C01820=1176.293,412.482,-85.837,-176.041,9.220,148.722
C01821=1176.297,412.234,-85.801,-176.041,9.217,148.722
C01822=1176.301,411.988,-85.765,-176.040,9.216,148.721
C01823=1176.305,411.740,-85.728,-176.040,9.215,148.721
C01824=1176.309,411.492,-85.693,-176.040,9.212,148.720
C01825=1176.313,411.245,-85.656,-176.040,9.210,148.719
C01826=1176.317,410.998,-85.621,-176.040,9.208,148.719
C01827=1176.321,410.750,-85.584,-176.039,9.206,148.718
C01828=1176.324,410.503,-85.548,-176.039,9.204,148.718
C01829=1176.328,410.255,-85.513,-176.039,9.202,148.717
C01830=1176.333,410.008,-85.476,-176.039,9.200,148.717
C01831=1176.336,409.761,-85.440,-176.038,9.198,148.716
C01832=1176.340,409.513,-85.404,-176.038,9.196,148.715
C01833=1176.344,409.266,-85.368,-176.038,9.195,148.715
C01834=1176.348,409.018,-85.332,-176.038,9.192,148.714
C01835=1176.352,408.771,-85.296,-176.038,9.191,148.714
C01836=1176.356,408.525,-85.260,-176.038,9.188,148.713
C01837=1176.360,408.277,-85.224,-176.038,9.186,148.713
C01838=1176.364,408.029,-85.188,-176.037,9.184,148.712
C01839=1176.368,407.782,-85.152,-176.037,9.182,148.711
C01840=1176.371,407.535,-85.116,-176.037,9.180,148.711
C01841=1176.375,407.287,-85.081,-176.037,9.178,148.710
C01842=1176.379,407.040,-85.044,-176.036,9.176,148.710
C01843=1176.383,406.792,-85.008,-176.036,9.174,148.709
C01844=1176.387,406.545,-84.972,-176.036,9.171,148.708
C01845=1176.391,406.297,-84.936,-176.036,9.170,148.708
C01846=1176.395,406.050,-84.900,-176.036,9.167,148.707
C01847=1176.399,405.803,-84.864,-176.036,9.166,148.707
C01848=1176.403,405.556,-84.829,-176.035,9.163,148.706
C01849=1176.407,405.308,-84.792,-176.035,9.161,148.705
C01850=1176.411,405.061,-84.756,-176.035,9.159,148.705
C01851=1176.414,404.813,-84.721,-176.035,9.157,148.704
C01852=1176.418,404.566,-84.684,-176.035,9.155,148.704
C01853=1176.422,404.319,-84.648,-176.034,9.153,148.703
C01854=1176.427,404.071,-84.612,-176.034,9.150,148.702
C01855=1176.430,403.823,-84.577,-176.034,9.148,148.702
C01856=1176.434,403.576,-84.541,-176.034,9.145,148.701
C01857=1176.439,403.329,-84.505,-176.034,9.144,148.701
C01858=1176.442,403.082,-84.469,-176.034,9.141,148.700
C01859=1176.446,402.835,-84.432,-176.034,9.139,148.699
C01860=1176.450,402.587,-84.397,-176.034,9.137,148.699
C01861=1176.454,402.340,-84.361,-176.033,9.135,148.698
C01862=1176.458,402.092,-84.325,-176.033,9.132,148.697
C01863=1176.461,401.845,-84.289,-176.033,9.130,148.697
C01864=1176.465,401.597,-84.253,-176.033,9.127,148.696
C01865=1176.470,401.350,-84.218,-176.032,9.126,148.695
C01866=1176.474,401.103,-84.182,-176.033,9.123,148.695
C01867=1176.477,400.855,-84.146,-176.033,9.121,148.694
C01868=1176.481,400.608,-84.110,-176.032,9.118,148.693
C01869=1176.485,400.361,-84.074,-176.033,9.116,148.693
C01870=1176.490,400.113,-84.038,-176.033,9.113,148.692
C01871=1176.493,399.865,-84.002,-176.032,9.111,148.691
C01872=1176.497,399.618,-83.966,-176.032,9.109,148.691
C01873=1176.502,399.371,-83.930,-176.032,9.107,148.690
C01874=1176.505,399.124,-83.895,-176.032,9.104,148.689
C01875=1176.509,398.876,-83.859,-176.032,9.102,148.689
C01876=1176.513,398.629,-83.823,-176.032,9.099,148.688
C01877=1176.517,398.382,-83.787,-176.032,9.097,148.688
C01878=1176.520,398.134,-83.751,-176.032,9.094,148.687
C01879=1176.525,397.886,-83.715,-176.032,9.092,148.686
C01880=1176.529,397.640,-83.680,-176.032,9.089,148.686
C01881=1176.533,397.392,-83.644,-176.031,9.087,148.685
C01882=1176.537,397.144,-83.608,-176.031,9.084,148.684
C01883=1176.540,396.897,-83.572,-176.032,9.082,148.684
C01884=1176.544,396.650,-83.536,-176.031,9.080,148.683
C01885=1176.548,396.402,-83.501,-176.031,9.077,148.682
C01886=1176.552,396.155,-83.465,-176.032,9.075,148.682
C01887=1176.556,395.908,-83.430,-176.032,9.071,148.681
C01888=1176.560,395.660,-83.394,-176.032,9.069,148.680
C01889=1176.564,395.412,-83.358,-176.032,9.066,148.679
C01890=1176.568,395.166,-83.322,-176.032,9.064,148.679
C01891=1176.571,394.918,-83.286,-176.032,9.061,148.678
C01892=1176.576,394.670,-83.250,-176.032,9.059,148.678
C01893=1176.580,394.423,-83.215,-176.031,9.056,148.677
C01894=1176.584,394.176,-83.179,-176.032,9.053,148.676
C01895=1176.587,393.928,-83.144,-176.032,9.051,148.675
C01896=1176.592,393.681,-83.107,-176.032,9.048,148.675
C01897=1176.596,393.433,-83.072,-176.032,9.045,148.674
C01898=1176.599,393.186,-83.036,-176.033,9.042,148.673
C01899=1176.603,392.939,-83.000,-176.032,9.040,148.673
C01900=1176.608,392.692,-82.964,-176.032,9.037,148.672
C01901=1176.611,392.444,-82.929,-176.033,9.034,148.671
C01902=1176.616,392.159,-82.888,-176.032,9.031,148.671
C01903=1176.620,391.875,-82.847,-176.033,9.028,148.670
C01904=1176.625,391.591,-82.806,-176.033,9.024,148.669
C01905=1176.629,391.307,-82.765,-176.034,9.021,148.668
C01906=1176.633,391.059,-82.729,-176.033,9.018,148.667
C01907=1176.637,390.811,-82.693,-176.034,9.016,148.667
C01908=1176.641,390.564,-82.658,-176.034,9.013,148.666
C01909=1176.645,390.317,-82.622,-176.034,9.010,148.665
C01910=1176.649,390.070,-82.587,-176.035,9.007,148.665
C01911=1176.653,389.822,-82.551,-176.035,9.005,148.664
C01912=1176.657,389.574,-82.515,-176.035,9.001,148.663
C01913=1176.661,389.327,-82.480,-176.036,8.998,148.663
C01914=1176.665,389.080,-82.444,-176.036,8.996,148.662
C01915=1176.668,388.832,-82.409,-176.037,8.992,148.662
C01916=1176.672,388.585,-82.373,-176.036,8.990,148.661
C01917=1176.677,388.337,-82.337,-176.037,8.986,148.660
C01918=1176.680,388.090,-82.302,-176.038,8.983,148.659
C01919=1176.684,387.843,-82.266,-176.037,8.981,148.659
C01920=1176.688,387.595,-82.231,-176.038,8.978,148.658
C01921=1176.692,387.348,-82.195,-176.039,8.974,148.657
C01922=1176.696,387.100,-82.159,-176.039,8.971,148.657
C01923=1176.700,386.853,-82.124,-176.039,8.969,148.656
C01924=1176.704,386.605,-82.089,-176.040,8.966,148.656
C01925=1176.708,386.358,-82.054,-176.041,8.962,148.655
C01926=1176.712,386.110,-82.018,-176.041,8.959,148.654
C01927=1176.715,385.863,-81.983,-176.042,8.956,148.653
C01928=1176.720,385.616,-81.947,-176.043,8.953,148.653
C01929=1176.724,385.368,-81.911,-176.043,8.949,148.652
C01930=1176.728,385.120,-81.876,-176.043,8.947,148.651
C01931=1176.731,384.873,-81.840,-176.044,8.944,148.651
C01932=1176.736,384.626,-81.805,-176.045,8.940,148.650
C01933=1176.740,384.378,-81.770,-176.045,8.937,148.650
C01934=1176.743,384.131,-81.735,-176.046,8.934,148.649
C01935=1176.747,383.883,-81.699,-176.047,8.931,148.648
C01936=1176.751,383.636,-81.664,-176.047,8.928,148.648
C01937=1176.756,383.388,-81.628,-176.048,8.924,148.647
C01938=1176.759,383.141,-81.592,-176.049,8.920,148.646
C01939=1176.764,382.894,-81.558,-176.050,8.917,148.646
C01940=1176.768,382.646,-81.522,-176.050,8.914,148.645
C01941=1176.771,382.399,-81.487,-176.051,8.911,148.644
C01942=1176.775,382.151,-81.451,-176.052,8.908,148.644
C01943=1176.779,381.904,-81.416,-176.053,8.905,148.643
C01944=1176.783,381.656,-81.381,-176.054,8.901,148.642
C01945=1176.787,381.409,-81.345,-176.055,8.897,148.642
C01946=1176.791,381.162,-81.310,-176.056,8.894,148.641
C01947=1176.795,380.914,-81.275,-176.056,8.891,148.641
C01948=1176.799,380.666,-81.240,-176.057,8.888,148.640
C01949=1176.803,380.419,-81.205,-176.059,8.884,148.639
C01950=1176.807,380.172,-81.169,-176.059,8.881,148.639
C01951=1176.811,379.924,-81.134,-176.060,8.878,148.638
C01952=1176.815,379.676,-81.098,-176.062,8.874,148.638
C01953=1176.819,379.429,-81.063,-176.062,8.871,148.637
C01954=1176.823,379.181,-81.028,-176.063,8.868,148.636
C01955=1176.827,378.934,-80.993,-176.065,8.864,148.636
C01956=1176.831,378.687,-80.957,-176.066,8.861,148.635
C01957=1176.835,378.439,-80.923,-176.067,8.857,148.635
C01958=1176.839,378.191,-80.887,-176.068,8.854,148.634
C01959=1176.843,377.944,-80.852,-176.069,8.850,148.633
C01960=1176.847,377.696,-80.817,-176.070,8.847,148.633
C01961=1176.851,377.449,-80.782,-176.071,8.844,148.632
C01962=1176.854,377.202,-80.748,-176.072,8.840,148.632
C01963=1176.858,376.954,-80.712,-176.074,8.836,148.631
C01964=1176.862,376.707,-80.677,-176.074,8.833,148.630
C01965=1176.866,376.459,-80.642,-176.076,8.829,148.630
C01966=1176.870,376.212,-80.607,-176.077,8.826,148.629
C01967=1176.875,375.964,-80.572,-176.078,8.822,148.629
C01968=1176.878,375.717,-80.537,-176.079,8.819,148.628
C01969=1176.882,375.469,-80.502,-176.081,8.816,148.628
C01970=1176.886,375.222,-80.467,-176.083,8.812,148.627
C01971=1176.890,374.974,-80.432,-176.083,8.809,148.626
C01972=1176.895,374.727,-80.397,-176.085,8.805,148.626
C01973=1176.899,374.479,-80.362,-176.086,8.802,148.625
C01974=1176.902,374.231,-80.326,-176.087,8.798,148.625
C01975=1176.906,373.984,-80.292,-176.089,8.794,148.624
C01976=1176.910,373.737,-80.257,-176.090,8.791,148.624
C01977=1176.914,373.489,-80.222,-176.092,8.788,148.623
C01978=1176.918,373.242,-80.187,-176.093,8.784,148.623
C01979=1176.922,372.994,-80.152,-176.095,8.780,148.622
C01980=1176.927,372.746,-80.117,-176.096,8.777,148.622
C01981=1176.930,372.499,-80.082,-176.097,8.773,148.621
C01982=1176.934,372.252,-80.048,-176.099,8.769,148.621
C01983=1176.938,372.004,-80.012,-176.101,8.766,148.620
C01984=1176.942,371.756,-79.978,-176.102,8.763,148.620
C01985=1176.946,371.509,-79.943,-176.104,8.759,148.619
C01986=1176.950,371.261,-79.908,-176.105,8.755,148.619
C01987=1176.954,371.014,-79.874,-176.107,8.752,148.618
C01988=1176.958,370.766,-79.839,-176.109,8.748,148.618
C01989=1176.962,370.519,-79.804,-176.110,8.744,148.617
C01990=1176.966,370.271,-79.769,-176.111,8.741,148.617
C01991=1176.971,370.023,-79.734,-176.113,8.738,148.616
C01992=1176.974,369.776,-79.699,-176.115,8.734,148.616
C01993=1176.978,369.529,-79.665,-176.116,8.730,148.615
C01994=1176.982,369.281,-79.630,-176.118,8.727,148.615
C01995=1176.987,369.033,-79.596,-176.120,8.723,148.614
C01996=1176.990,368.786,-79.561,-176.122,8.719,148.614
C01997=1176.994,368.539,-79.526,-176.123,8.715,148.613
C01998=1176.998,368.291,-79.491,-176.125,8.712,148.613
C01999=1177.002,368.043,-79.458,-176.127,8.708,148.612
C02000=1177.006,367.795,-79.423,-176.129,8.705,148.612
C02001=1177.010,367.548,-79.388,-176.130,8.702,148.612
C02002=1177.014,367.300,-79.353,-176.132,8.698,148.611
C02003=1177.018,367.053,-79.319,-176.134,8.695,148.611
C02004=1177.022,366.805,-79.284,-176.136,8.691,148.610
C02005=1177.026,366.558,-79.250,-176.137,8.687,148.610
C02006=1177.030,366.276,-79.210,-176.140,8.683,148.609
C02007=1177.035,365.994,-79.171,-176.142,8.679,148.609
C02008=1177.040,365.712,-79.131,-176.144,8.675,148.609
C02009=1177.044,365.431,-79.093,-176.146,8.670,148.608
C02010=1177.048,365.182,-79.058,-176.148,8.667,148.608
C02011=1177.052,364.936,-79.024,-176.150,8.663,148.607
C02012=1177.056,364.688,-78.989,-176.152,8.660,148.607
C02013=1177.060,364.440,-78.955,-176.154,8.656,148.606
C02014=1177.064,364.193,-78.921,-176.156,8.652,148.606
C02015=1177.068,363.945,-78.886,-176.158,8.649,148.606
C02016=1177.072,363.698,-78.852,-176.160,8.645,148.605
C02017=1177.076,363.449,-78.818,-176.162,8.642,148.605
C02018=1177.080,363.202,-78.784,-176.163,8.638,148.604
C02019=1177.084,362.954,-78.749,-176.166,8.635,148.604
C02020=1177.089,362.707,-78.715,-176.167,8.631,148.604
C02021=1177.092,362.460,-78.681,-176.169,8.628,148.603
C02022=1177.096,362.211,-78.646,-176.171,8.624,148.603
C02023=1177.100,361.964,-78.612,-176.174,8.620,148.603
C02024=1177.104,361.716,-78.577,-176.176,8.616,148.602
C02025=1177.108,361.469,-78.543,-176.178,8.613,148.602
C02026=1177.113,361.222,-78.509,-176.180,8.609,148.602
C02027=1177.116,360.973,-78.475,-176.182,8.606,148.601
C02028=1177.121,360.726,-78.441,-176.184,8.602,148.601
C02029=1177.124,360.479,-78.407,-176.186,8.599,148.600
C02030=1177.128,360.231,-78.373,-176.188,8.595,148.600
C02031=1177.132,359.983,-78.338,-176.190,8.591,148.600
C02032=1177.136,359.735,-78.305,-176.193,8.588,148.600
C02033=1177.140,359.488,-78.270,-176.195,8.584,148.599
C02034=1177.144,359.241,-78.237,-176.197,8.581,148.599
C02035=1177.148,358.992,-78.202,-176.199,8.577,148.598
C02036=1177.152,358.745,-78.169,-176.201,8.574,148.598
C02037=1177.156,358.498,-78.135,-176.203,8.570,148.598
C02038=1177.160,358.249,-78.100,-176.206,8.566,148.598
C02039=1177.164,358.002,-78.067,-176.208,8.563,148.597
C02040=1177.169,357.754,-78.032,-176.210,8.559,148.597
C02041=1177.173,357.507,-77.998,-176.212,8.556,148.597
C02042=1177.176,357.259,-77.965,-176.214,8.552,148.596
C02043=1177.181,357.011,-77.930,-176.216,8.549,148.596
C02044=1177.185,356.764,-77.896,-176.218,8.546,148.596
C02045=1177.188,356.516,-77.863,-176.221,8.541,148.595
C02046=1177.193,356.268,-77.828,-176.223,8.538,148.595
C02047=1177.197,356.021,-77.795,-176.225,8.535,148.595
C02048=1177.201,355.774,-77.761,-176.227,8.531,148.594
C02049=1177.205,355.525,-77.727,-176.229,8.528,148.594
C02050=1177.209,355.278,-77.693,-176.232,8.524,148.594
C02051=1177.213,355.030,-77.660,-176.235,8.520,148.594
C02052=1177.217,354.783,-77.626,-176.236,8.517,148.593
C02053=1177.221,354.534,-77.592,-176.239,8.513,148.593
C02054=1177.225,354.287,-77.558,-176.241,8.510,148.593
C02055=1177.229,354.039,-77.525,-176.243,8.506,148.592
C02056=1177.234,353.792,-77.491,-176.245,8.503,148.592
C02057=1177.237,353.543,-77.457,-176.247,8.500,148.592
C02058=1177.241,353.296,-77.423,-176.250,8.496,148.592
C02059=1177.245,353.049,-77.390,-176.252,8.492,148.591
C02060=1177.250,352.801,-77.356,-176.254,8.489,148.591
C02061=1177.254,352.553,-77.323,-176.256,8.485,148.591
C02062=1177.257,352.305,-77.289,-176.259,8.482,148.591
C02063=1177.261,352.058,-77.255,-176.261,8.479,148.590
C02064=1177.265,351.810,-77.222,-176.263,8.475,148.590
C02065=1177.270,351.562,-77.188,-176.265,8.472,148.590
C02066=1177.274,351.315,-77.155,-176.268,8.468,148.589
C02067=1177.278,351.067,-77.121,-176.270,8.464,148.589
C02068=1177.282,350.819,-77.088,-176.272,8.461,148.589
C02069=1177.286,350.571,-77.055,-176.275,8.458,148.589
C02070=1177.290,350.324,-77.021,-176.277,8.455,148.589
C02071=1177.294,350.076,-76.988,-176.279,8.451,148.588
C02072=1177.299,349.828,-76.954,-176.281,8.448,148.588
C02073=1177.303,349.581,-76.921,-176.283,8.444,148.588
C02074=1177.307,349.333,-76.887,-176.286,8.440,148.587
C02075=1177.310,349.085,-76.853,-176.288,8.437,148.587
C02076=1177.314,348.837,-76.820,-176.291,8.434,148.587
C02077=1177.318,348.590,-76.787,-176.293,8.430,148.587
C02078=1177.323,348.342,-76.754,-176.295,8.427,148.587
C02079=1177.326,348.095,-76.720,-176.298,8.424,148.586
C02080=1177.331,347.847,-76.687,-176.300,8.420,148.586
C02081=1177.335,347.599,-76.654,-176.302,8.417,148.586
C02082=1177.339,347.352,-76.621,-176.304,8.414,148.586
C02083=1177.343,347.104,-76.587,-176.307,8.410,148.585
C02084=1177.347,346.856,-76.554,-176.309,8.406,148.585
C02085=1177.351,346.608,-76.521,-176.311,8.403,148.585
C02086=1177.355,346.360,-76.488,-176.314,8.399,148.585
C02087=1177.359,346.112,-76.454,-176.316,8.396,148.584
C02088=1177.363,345.864,-76.421,-176.318,8.393,148.584
C02089=1177.367,345.617,-76.388,-176.320,8.389,148.584
C02090=1177.371,345.369,-76.355,-176.323,8.386,148.584
C02091=1177.375,345.121,-76.322,-176.325,8.383,148.584
C02092=1177.380,344.874,-76.289,-176.328,8.380,148.584
C02093=1177.384,344.626,-76.255,-176.330,8.376,148.583
C02094=1177.388,344.378,-76.222,-176.333,8.372,148.583
C02095=1177.392,344.130,-76.189,-176.335,8.369,148.583
C02096=1177.396,343.883,-76.156,-176.337,8.366,148.583
C02097=1177.400,343.635,-76.123,-176.340,8.362,148.582
C02098=1177.404,343.387,-76.090,-176.342,8.359,148.582
C02099=1177.409,343.139,-76.057,-176.344,8.356,148.582
C02100=1177.413,342.891,-76.024,-176.346,8.352,148.582
C02101=1177.417,342.643,-75.991,-176.349,8.349,148.582
C02102=1177.421,342.396,-75.958,-176.351,8.346,148.581
C02103=1177.425,342.148,-75.925,-176.353,8.343,148.581
C02104=1177.429,341.900,-75.892,-176.355,8.339,148.581
C02105=1177.433,341.652,-75.860,-176.358,8.335,148.581
C02106=1177.437,341.404,-75.826,-176.361,8.332,148.581
C02107=1177.442,341.157,-75.793,-176.363,8.329,148.580
C02108=1177.446,340.909,-75.760,-176.366,8.325,148.580
C02109=1177.450,340.661,-75.727,-176.368,8.322,148.580
C02110=1177.455,340.382,-75.691,-176.370,8.319,148.580
C02111=1177.459,340.102,-75.654,-176.373,8.315,148.580
C02112=1177.464,339.824,-75.617,-176.376,8.311,148.579
C02113=1177.469,339.545,-75.580,-176.378,8.308,148.579
C02114=1177.472,339.298,-75.547,-176.381,8.304,148.579
C02115=1177.477,339.049,-75.515,-176.383,8.301,148.579
C02116=1177.481,338.801,-75.482,-176.385,8.298,148.579
C02117=1177.485,338.554,-75.449,-176.388,8.294,148.578
C02118=1177.489,338.306,-75.417,-176.390,8.290,148.578
C02119=1177.493,338.058,-75.384,-176.393,8.287,148.578
C02120=1177.497,337.810,-75.351,-176.395,8.284,148.578
C02121=1177.501,337.562,-75.318,-176.398,8.281,148.578
C02122=1177.505,337.314,-75.285,-176.400,8.277,148.578
C02123=1177.509,337.066,-75.253,-176.403,8.274,148.578
C02124=1177.514,336.819,-75.220,-176.405,8.271,148.577
C02125=1177.518,336.571,-75.188,-176.407,8.268,148.577
C02126=1177.522,336.323,-75.155,-176.409,8.264,148.577
C02127=1177.526,336.075,-75.123,-176.412,8.261,148.577
C02128=1177.530,335.828,-75.090,-176.414,8.258,148.577
C02129=1177.534,335.579,-75.058,-176.417,8.255,148.576
C02130=1177.538,335.331,-75.025,-176.419,8.251,148.576
C02131=1177.542,335.083,-74.993,-176.421,8.248,148.576
C02132=1177.547,334.836,-74.961,-176.424,8.245,148.576
C02133=1177.550,334.588,-74.928,-176.426,8.242,148.576
C02134=1177.555,334.340,-74.896,-176.429,8.239,148.576
C02135=1177.559,334.092,-74.862,-176.431,8.236,148.576
C02136=1177.563,333.844,-74.831,-176.433,8.232,148.575
C02137=1177.567,333.596,-74.798,-176.436,8.228,148.575
C02138=1177.571,333.349,-74.766,-176.439,8.225,148.575
C02139=1177.576,333.101,-74.734,-176.441,8.222,148.575
C02140=1177.579,332.853,-74.702,-176.444,8.219,148.575
C02141=1177.583,332.605,-74.669,-176.446,8.215,148.575
C02142=1177.588,332.357,-74.636,-176.449,8.212,148.575
C02143=1177.592,332.109,-74.605,-176.451,8.209,148.574
C02144=1177.596,331.862,-74.571,-176.453,8.206,148.574
C02145=1177.600,331.614,-74.540,-176.456,8.203,148.574
C02146=1177.604,331.365,-74.507,-176.458,8.199,148.574
C02147=1177.609,331.118,-74.476,-176.460,8.196,148.574
C02148=1177.613,330.870,-74.443,-176.463,8.193,148.574
C02149=1177.617,330.622,-74.411,-176.465,8.190,148.574
C02150=1177.620,330.374,-74.379,-176.468,8.186,148.573
C02151=1177.625,330.126,-74.347,-176.470,8.183,148.573
C02152=1177.629,329.878,-74.315,-176.473,8.180,148.573
C02153=1177.634,329.630,-74.283,-176.475,8.177,148.573
C02154=1177.637,329.383,-74.250,-176.478,8.174,148.573
C02155=1177.642,329.135,-74.218,-176.480,8.170,148.573
C02156=1177.646,328.887,-74.186,-176.483,8.167,148.573
C02157=1177.650,328.639,-74.154,-176.485,8.164,148.572
C02158=1177.654,328.391,-74.122,-176.487,8.161,148.572
C02159=1177.658,328.143,-74.090,-176.490,8.158,148.572
C02160=1177.663,327.895,-74.058,-176.492,8.155,148.572
C02161=1177.666,327.647,-74.026,-176.494,8.151,148.572
C02162=1177.671,327.400,-73.995,-176.497,8.148,148.572
C02163=1177.675,327.151,-73.962,-176.499,8.145,148.572
C02164=1177.679,326.903,-73.930,-176.502,8.142,148.572
C02165=1177.683,326.656,-73.899,-176.504,8.139,148.571
C02166=1177.687,326.407,-73.866,-176.507,8.136,148.571
C02167=1177.691,326.159,-73.834,-176.509,8.132,148.571
C02168=1177.696,325.912,-73.803,-176.512,8.129,148.571
C02169=1177.700,325.664,-73.771,-176.514,8.126,148.571
C02170=1177.704,325.416,-73.739,-176.517,8.123,148.571
C02171=1177.708,325.168,-73.707,-176.519,8.120,148.571
C02172=1177.712,324.920,-73.675,-176.522,8.116,148.571
C02173=1177.717,324.673,-73.643,-176.524,8.113,148.571
C02174=1177.720,324.425,-73.611,-176.527,8.110,148.570
C02175=1177.724,324.176,-73.580,-176.529,8.107,148.570
C02176=1177.729,323.928,-73.548,-176.532,8.104,148.570
C02177=1177.733,323.680,-73.516,-176.534,8.101,148.570
C02178=1177.737,323.432,-73.485,-176.537,8.098,148.570
C02179=1177.741,323.185,-73.453,-176.539,8.094,148.570
C02180=1177.745,322.937,-73.421,-176.542,8.091,148.570
C02181=1177.750,322.689,-73.390,-176.544,8.088,148.570
C02182=1177.754,322.441,-73.358,-176.547,8.085,148.570
C02183=1177.758,322.193,-73.326,-176.549,8.082,148.569
C02184=1177.762,321.945,-73.295,-176.552,8.079,148.569
C02185=1177.766,321.697,-73.264,-176.554,8.075,148.569
C02186=1177.770,321.449,-73.232,-176.557,8.072,148.569
C02187=1177.775,321.201,-73.200,-176.559,8.069,148.569
C02188=1177.779,320.952,-73.169,-176.562,8.066,148.569
C02189=1177.783,320.705,-73.137,-176.564,8.063,148.569
C02190=1177.787,320.457,-73.105,-176.567,8.060,148.569
C02191=1177.791,320.209,-73.074,-176.569,8.056,148.569
C02192=1177.795,319.961,-73.043,-176.572,8.053,148.569
C02193=1177.799,319.713,-73.011,-176.574,8.050,148.569
C02194=1177.803,319.465,-72.980,-176.577,8.047,148.569
C02195=1177.808,319.217,-72.948,-176.579,8.044,148.569
C02196=1177.812,318.969,-72.917,-176.582,8.041,148.568
C02197=1177.817,318.721,-72.885,-176.584,8.038,148.568
C02198=1177.820,318.473,-72.853,-176.586,8.035,148.568
C02199=1177.825,318.225,-72.823,-176.589,8.032,148.568
C02200=1177.829,317.977,-72.791,-176.591,8.028,148.568
C02201=1177.833,317.729,-72.760,-176.594,8.025,148.568
C02202=1177.837,317.481,-72.728,-176.596,8.022,148.568
C02203=1177.842,317.233,-72.697,-176.599,8.019,148.568
C02204=1177.845,316.985,-72.666,-176.602,8.016,148.568
C02205=1177.850,316.737,-72.635,-176.604,8.013,148.568
C02206=1177.854,316.489,-72.603,-176.607,8.010,148.568
C02207=1177.858,316.241,-72.572,-176.609,8.006,148.567
C02208=1177.862,315.993,-72.541,-176.612,8.003,148.567
C02209=1177.867,315.745,-72.510,-176.614,8.000,148.567
C02210=1177.871,315.497,-72.479,-176.617,7.997,148.567
C02211=1177.875,315.249,-72.447,-176.620,7.994,148.567
C02212=1177.880,315.001,-72.416,-176.621,7.992,148.567
C02213=1177.884,314.753,-72.385,-176.624,7.989,148.567
C02214=1177.888,314.476,-72.350,-176.627,7.984,148.567
C02215=1177.893,314.199,-72.315,-176.630,7.981,148.567
C02216=1177.897,313.922,-72.281,-176.633,7.978,148.567
C02217=1177.903,313.646,-72.246,-176.635,7.974,148.567
C02218=1177.906,313.398,-72.216,-176.638,7.971,148.567
C02219=1177.910,313.150,-72.184,-176.641,7.968,148.567
C02220=1177.914,312.902,-72.153,-176.643,7.965,148.566
C02221=1177.919,312.654,-72.123,-176.646,7.962,148.567
C02222=1177.924,312.406,-72.092,-176.648,7.959,148.567
C02223=1177.927,312.158,-72.060,-176.651,7.956,148.566
C02224=1177.932,311.910,-72.029,-176.653,7.953,148.566
C02225=1177.935,311.661,-71.999,-176.656,7.949,148.566
C02226=1177.940,311.413,-71.968,-176.658,7.946,148.566
C02227=1177.944,311.166,-71.937,-176.661,7.943,148.566
C02228=1177.948,310.917,-71.905,-176.663,7.940,148.566
C02229=1177.953,310.670,-71.874,-176.665,7.938,148.566
C02230=1177.957,310.422,-71.844,-176.668,7.935,148.566
C02231=1177.961,310.173,-71.813,-176.670,7.932,148.566
C02232=1177.965,309.925,-71.782,-176.673,7.929,148.566
C02233=1177.970,309.677,-71.752,-176.676,7.926,148.566
C02234=1177.974,309.429,-71.721,-176.678,7.922,148.566
C02235=1177.978,309.181,-71.690,-176.681,7.919,148.566
C02236=1177.982,308.933,-71.660,-176.684,7.916,148.566
C02237=1177.986,308.684,-71.628,-176.686,7.913,148.566
C02238=1177.991,308.436,-71.598,-176.689,7.910,148.566
C02239=1177.995,308.189,-71.568,-176.691,7.907,148.566
C02240=1177.999,307.941,-71.537,-176.694,7.904,148.565
C02241=1178.003,307.692,-71.506,-176.696,7.901,148.565
C02242=1178.007,307.444,-71.475,-176.699,7.898,148.565
C02243=1178.012,307.197,-71.445,-176.701,7.895,148.565
C02244=1178.017,306.949,-71.414,-176.703,7.892,148.565
C02245=1178.020,306.700,-71.383,-176.706,7.889,148.565
C02246=1178.024,306.452,-71.353,-176.709,7.886,148.565
C02247=1178.029,306.204,-71.322,-176.711,7.883,148.565
C02248=1178.033,305.957,-71.292,-176.714,7.880,148.565
C02249=1178.037,305.708,-71.261,-176.717,7.877,148.565
C02250=1178.042,305.459,-71.231,-176.719,7.874,148.565
C02251=1178.046,305.212,-71.200,-176.722,7.871,148.565
C02252=1178.050,304.964,-71.170,-176.724,7.868,148.565
C02253=1178.054,304.715,-71.139,-176.727,7.865,148.565
C02254=1178.058,304.468,-71.108,-176.729,7.862,148.565
C02255=1178.063,304.219,-71.078,-176.732,7.859,148.565
C02256=1178.067,303.971,-71.048,-176.734,7.856,148.565
C02257=1178.072,303.723,-71.017,-176.737,7.853,148.565
C02258=1178.075,303.475,-70.987,-176.739,7.850,148.565
C02259=1178.080,303.227,-70.956,-176.742,7.847,148.565
C02260=1178.084,302.979,-70.927,-176.745,7.844,148.565
C02261=1178.088,302.731,-70.896,-176.747,7.841,148.565
C02262=1178.093,302.483,-70.865,-176.750,7.838,148.565
C02263=1178.097,302.235,-70.836,-176.752,7.835,148.565
C02264=1178.101,301.986,-70.804,-176.755,7.832,148.565
C02265=1178.105,301.738,-70.774,-176.757,7.829,148.565
C02266=1178.110,301.490,-70.744,-176.760,7.826,148.565
C02267=1178.114,301.242,-70.714,-176.762,7.823,148.565
C02268=1178.118,300.994,-70.684,-176.765,7.820,148.565
C02269=1178.123,300.746,-70.654,-176.767,7.817,148.564
C02270=1178.126,300.497,-70.623,-176.770,7.814,148.564
C02271=1178.131,300.249,-70.593,-176.773,7.811,148.564
C02272=1178.135,300.001,-70.563,-176.775,7.808,148.565
C02273=1178.140,299.753,-70.533,-176.778,7.805,148.564
C02274=1178.143,299.505,-70.503,-176.780,7.803,148.564
C02275=1178.148,299.257,-70.472,-176.783,7.800,148.564
C02276=1178.152,299.009,-70.443,-176.785,7.797,148.564
C02277=1178.156,298.761,-70.413,-176.788,7.794,148.564
C02278=1178.161,298.513,-70.382,-176.790,7.790,148.564
C02279=1178.164,298.264,-70.352,-176.793,7.787,148.564
C02280=1178.168,298.016,-70.322,-176.796,7.784,148.564
C02281=1178.173,297.767,-70.292,-176.799,7.781,148.564
C02282=1178.177,297.520,-70.262,-176.801,7.778,148.564
C02283=1178.182,297.271,-70.232,-176.803,7.776,148.564
C02284=1178.186,297.023,-70.202,-176.806,7.773,148.564
C02285=1178.190,296.775,-70.173,-176.808,7.770,148.564
C02286=1178.194,296.528,-70.142,-176.811,7.767,148.564
C02287=1178.199,296.279,-70.112,-176.814,7.764,148.564
C02288=1178.203,296.031,-70.083,-176.816,7.761,148.564
C02289=1178.207,295.783,-70.053,-176.819,7.758,148.564
C02290=1178.212,295.535,-70.023,-176.821,7.756,148.564
C02291=1178.216,295.286,-69.993,-176.824,7.753,148.564
C02292=1178.220,295.039,-69.963,-176.827,7.750,148.564
C02293=1178.224,294.790,-69.934,-176.829,7.746,148.564
C02294=1178.229,294.542,-69.904,-176.832,7.743,148.564
C02295=1178.233,294.293,-69.874,-176.834,7.740,148.564
C02296=1178.237,294.046,-69.844,-176.837,7.737,148.564
C02297=1178.241,293.798,-69.815,-176.840,7.734,148.564
C02298=1178.246,293.549,-69.784,-176.842,7.732,148.564
C02299=1178.251,293.301,-69.755,-176.844,7.729,148.564
C02300=1178.254,293.053,-69.725,-176.847,7.726,148.564
C02301=1178.259,292.805,-69.695,-176.850,7.723,148.564
C02302=1178.263,292.557,-69.666,-176.852,7.720,148.564
C02303=1178.267,292.308,-69.636,-176.855,7.717,148.564
C02304=1178.272,292.060,-69.606,-176.857,7.715,148.564
C02305=1178.276,291.811,-69.577,-176.860,7.712,148.564
C02306=1178.280,291.564,-69.547,-176.862,7.708,148.564
C02307=1178.284,291.316,-69.517,-176.865,7.705,148.564
C02308=1178.288,291.067,-69.488,-176.868,7.702,148.564
C02309=1178.292,290.819,-69.458,-176.870,7.700,148.564
C02310=1178.297,290.571,-69.429,-176.873,7.697,148.564
C02311=1178.302,290.322,-69.399,-176.875,7.694,148.564
C02312=1178.306,290.074,-69.369,-176.878,7.691,148.564
C02313=1178.310,289.826,-69.340,-176.880,7.688,148.564
C02314=1178.314,289.577,-69.311,-176.883,7.685,148.564
C02315=1178.318,289.329,-69.281,-176.886,7.682,148.564
C02316=1178.322,289.081,-69.252,-176.888,7.679,148.564
C02317=1178.327,288.833,-69.223,-176.891,7.677,148.564
C02318=1178.332,288.558,-69.189,-176.894,7.673,148.564
C02319=1178.336,288.283,-69.157,-176.897,7.670,148.564
C02320=1178.342,288.009,-69.125,-176.899,7.667,148.564
C02321=1178.346,287.734,-69.092,-176.902,7.664,148.564
C02322=1178.350,287.486,-69.063,-176.905,7.661,148.564
C02323=1178.354,287.238,-69.033,-176.908,7.658,148.565
C02324=1178.359,286.990,-69.005,-176.910,7.655,148.565
C02325=1178.363,286.741,-68.976,-176.913,7.652,148.565
C02326=1178.367,286.493,-68.946,-176.915,7.650,148.564
C02327=1178.372,286.245,-68.917,-176.917,7.647,148.564
C02328=1178.376,285.996,-68.887,-176.920,7.644,148.565
C02329=1178.380,285.748,-68.858,-176.923,7.641,148.565
C02330=1178.384,285.500,-68.828,-176.926,7.638,148.565
C02331=1178.389,285.252,-68.800,-176.928,7.636,148.565
C02332=1178.393,285.004,-68.770,-176.931,7.633,148.565
C02333=1178.398,284.755,-68.741,-176.933,7.630,148.565
C02334=1178.402,284.507,-68.712,-176.936,7.627,148.565
C02335=1178.406,284.258,-68.683,-176.939,7.624,148.565
C02336=1178.411,284.011,-68.654,-176.941,7.622,148.565
C02337=1178.415,283.762,-68.624,-176.944,7.619,148.565
C02338=1178.419,283.514,-68.595,-176.946,7.616,148.565
C02339=1178.423,283.265,-68.567,-176.949,7.612,148.565
C02340=1178.428,283.018,-68.538,-176.951,7.609,148.565
C02341=1178.432,282.770,-68.508,-176.954,7.607,148.565
C02342=1178.437,282.521,-68.479,-176.956,7.604,148.565
C02343=1178.441,282.272,-68.450,-176.959,7.601,148.565
C02344=1178.445,282.024,-68.421,-176.962,7.598,148.565
C02345=1178.449,281.776,-68.393,-176.964,7.595,148.565
C02346=1178.453,281.528,-68.363,-176.967,7.593,148.565
C02347=1178.458,281.279,-68.335,-176.969,7.590,148.565
C02348=1178.463,281.032,-68.305,-176.972,7.587,148.565
C02349=1178.467,280.783,-68.277,-176.975,7.584,148.565
C02350=1178.471,280.535,-68.248,-176.978,7.581,148.565
C02351=1178.475,280.286,-68.219,-176.980,7.579,148.565
C02352=1178.480,280.038,-68.190,-176.982,7.576,148.565
C02353=1178.484,279.789,-68.161,-176.985,7.573,148.565
C02354=1178.488,279.541,-68.132,-176.988,7.570,148.565
C02355=1178.492,279.293,-68.104,-176.990,7.568,148.566
C02356=1178.497,279.045,-68.075,-176.993,7.565,148.566
C02357=1178.502,278.796,-68.046,-176.996,7.562,148.566
C02358=1178.505,278.548,-68.017,-176.998,7.559,148.566
C02359=1178.510,278.300,-67.989,-177.001,7.556,148.566
C02360=1178.514,278.052,-67.959,-177.003,7.554,148.566
C02361=1178.518,277.803,-67.931,-177.006,7.551,148.566
C02362=1178.523,277.556,-67.902,-177.009,7.548,148.566
C02363=1178.527,277.307,-67.873,-177.011,7.545,148.566
C02364=1178.531,277.058,-67.845,-177.014,7.543,148.566
C02365=1178.536,276.810,-67.816,-177.016,7.540,148.566
C02366=1178.540,276.562,-67.787,-177.019,7.537,148.566
C02367=1178.544,276.313,-67.759,-177.022,7.534,148.566
C02368=1178.549,276.065,-67.730,-177.024,7.532,148.566
C02369=1178.553,275.817,-67.701,-177.027,7.529,148.566
C02370=1178.557,275.568,-67.673,-177.029,7.526,148.566
C02371=1178.562,275.320,-67.644,-177.032,7.523,148.566
C02372=1178.566,275.072,-67.616,-177.034,7.521,148.566
C02373=1178.571,274.824,-67.588,-177.037,7.518,148.566
C02374=1178.575,274.575,-67.559,-177.040,7.515,148.566
C02375=1178.579,274.326,-67.531,-177.043,7.512,148.567
C02376=1178.584,274.079,-67.502,-177.045,7.509,148.567
C02377=1178.588,273.830,-67.473,-177.047,7.506,148.567
C02378=1178.593,273.582,-67.445,-177.050,7.503,148.567
C02379=1178.596,273.333,-67.417,-177.053,7.501,148.567
C02380=1178.601,273.084,-67.388,-177.055,7.498,148.567
C02381=1178.605,272.837,-67.360,-177.058,7.495,148.567
C02382=1178.609,272.588,-67.331,-177.061,7.492,148.567
C02383=1178.614,272.340,-67.303,-177.063,7.489,148.567
C02384=1178.618,272.091,-67.274,-177.065,7.487,148.567
C02385=1178.623,271.844,-67.247,-177.068,7.484,148.567
C02386=1178.627,271.595,-67.218,-177.071,7.481,148.567
C02387=1178.631,271.347,-67.190,-177.073,7.479,148.567
C02388=1178.636,271.098,-67.161,-177.076,7.476,148.567
C02389=1178.640,270.849,-67.133,-177.079,7.474,148.568
C02390=1178.645,270.601,-67.105,-177.082,7.471,148.568
C02391=1178.648,270.353,-67.077,-177.084,7.468,148.568
C02392=1178.653,270.105,-67.049,-177.087,7.465,148.568
C02393=1178.657,269.856,-67.020,-177.089,7.462,148.568
C02394=1178.662,269.608,-66.992,-177.092,7.459,148.568
C02395=1178.666,269.359,-66.964,-177.094,7.457,148.568
C02396=1178.671,269.111,-66.936,-177.097,7.454,148.568
C02397=1178.674,268.863,-66.908,-177.100,7.451,148.568
C02398=1178.679,268.614,-66.879,-177.102,7.449,148.568
C02399=1178.683,268.366,-66.851,-177.105,7.446,148.568
C02400=1178.688,268.118,-66.823,-177.107,7.443,148.568
C02401=1178.692,267.869,-66.795,-177.110,7.441,148.568
C02402=1178.696,267.621,-66.767,-177.113,7.438,148.568
C02403=1178.701,267.373,-66.739,-177.116,7.435,148.569
C02404=1178.705,267.124,-66.711,-177.118,7.432,148.569
C02405=1178.710,266.876,-66.683,-177.120,7.430,148.569
C02406=1178.714,266.627,-66.655,-177.123,7.427,148.569
C02407=1178.719,266.379,-66.627,-177.126,7.424,148.569
C02408=1178.722,266.131,-66.599,-177.128,7.422,148.569
C02409=1178.727,265.882,-66.570,-177.131,7.419,148.569
C02410=1178.732,265.634,-66.543,-177.134,7.416,148.569
C02411=1178.736,265.385,-66.515,-177.136,7.414,148.569
C02412=1178.740,265.138,-66.487,-177.139,7.411,148.569
C02413=1178.745,264.889,-66.459,-177.142,7.408,148.569
C02414=1178.749,264.640,-66.432,-177.144,7.406,148.569
C02415=1178.753,264.392,-66.403,-177.147,7.403,148.570
C02416=1178.757,264.144,-66.376,-177.149,7.400,148.570
C02417=1178.763,263.895,-66.348,-177.152,7.397,148.570
C02418=1178.767,263.646,-66.320,-177.154,7.395,148.570
C02419=1178.771,263.398,-66.292,-177.157,7.393,148.570
C02420=1178.776,263.150,-66.265,-177.160,7.390,148.570
C02421=1178.779,262.901,-66.237,-177.162,7.387,148.570
C02422=1178.785,262.629,-66.207,-177.165,7.384,148.570
C02423=1178.789,262.355,-66.176,-177.168,7.382,148.570
C02424=1178.794,262.082,-66.145,-177.171,7.379,148.570
C02425=1178.799,261.809,-66.115,-177.174,7.376,148.571
C02426=1178.803,261.561,-66.087,-177.176,7.373,148.571
C02427=1178.808,261.312,-66.060,-177.179,7.370,148.571
C02428=1178.812,261.064,-66.032,-177.181,7.368,148.571
C02429=1178.816,260.815,-66.005,-177.185,7.365,148.571
C02430=1178.821,260.567,-65.976,-177.187,7.362,148.571
C02431=1178.826,260.319,-65.949,-177.189,7.360,148.571
C02432=1178.830,260.071,-65.921,-177.192,7.357,148.571
C02433=1178.834,259.822,-65.894,-177.195,7.354,148.571
C02434=1178.839,259.574,-65.866,-177.197,7.352,148.571
C02435=1178.843,259.325,-65.839,-177.200,7.349,148.572
C02436=1178.847,259.077,-65.811,-177.203,7.346,148.572
C02437=1178.852,258.828,-65.784,-177.205,7.344,148.572
C02438=1178.856,258.580,-65.756,-177.208,7.341,148.572
C02439=1178.860,258.331,-65.729,-177.210,7.339,148.572
C02440=1178.865,258.083,-65.702,-177.213,7.336,148.572
C02441=1178.869,257.835,-65.674,-177.216,7.333,148.572
C02442=1178.874,257.586,-65.647,-177.218,7.331,148.572
C02443=1178.877,257.338,-65.619,-177.221,7.328,148.572
C02444=1178.882,257.089,-65.592,-177.224,7.325,148.572
C02445=1178.887,256.841,-65.564,-177.226,7.323,148.573
C02446=1178.891,256.593,-65.537,-177.229,7.320,148.573
C02447=1178.895,256.344,-65.509,-177.232,7.318,148.573
C02448=1178.900,256.095,-65.482,-177.234,7.315,148.573
C02449=1178.904,255.847,-65.455,-177.237,7.312,148.573
C02450=1178.909,255.599,-65.427,-177.239,7.311,148.573
C02451=1178.913,255.350,-65.400,-177.242,7.308,148.573
C02452=1178.918,255.101,-65.373,-177.245,7.305,148.573
C02453=1178.922,254.852,-65.346,-177.247,7.302,148.574
C02454=1178.927,254.605,-65.318,-177.250,7.299,148.574
C02455=1178.931,254.356,-65.291,-177.252,7.298,148.574
C02456=1178.936,254.108,-65.264,-177.255,7.295,148.574
C02457=1178.939,253.859,-65.237,-177.258,7.292,148.574
C02458=1178.944,253.610,-65.210,-177.260,7.290,148.574
C02459=1178.948,253.362,-65.182,-177.263,7.287,148.574
C02460=1178.953,253.114,-65.155,-177.266,7.284,148.574
C02461=1178.957,252.865,-65.128,-177.268,7.282,148.575
C02462=1178.962,252.616,-65.101,-177.271,7.279,148.575
C02463=1178.966,252.368,-65.074,-177.274,7.277,148.575
C02464=1178.970,252.119,-65.047,-177.276,7.274,148.575
C02465=1178.975,251.871,-65.020,-177.279,7.271,148.575
C02466=1178.979,251.622,-64.993,-177.281,7.269,148.575
C02467=1178.984,251.374,-64.966,-177.284,7.266,148.575
C02468=1178.989,251.125,-64.939,-177.287,7.264,148.575
C02469=1178.992,250.877,-64.912,-177.289,7.261,148.576
C02470=1178.997,250.628,-64.885,-177.292,7.259,148.576
C02471=1179.001,250.380,-64.858,-177.295,7.256,148.576
C02472=1179.006,250.131,-64.831,-177.298,7.253,148.576
C02473=1179.010,249.883,-64.804,-177.300,7.251,148.576
C02474=1179.015,249.634,-64.777,-177.303,7.249,148.576
C02475=1179.019,249.386,-64.750,-177.305,7.246,148.576
C02476=1179.024,249.137,-64.723,-177.308,7.243,148.577
C02477=1179.028,248.889,-64.697,-177.311,7.241,148.577
C02478=1179.032,248.641,-64.670,-177.313,7.239,148.577
C02479=1179.037,248.392,-64.643,-177.316,7.236,148.577
C02480=1179.041,248.143,-64.615,-177.318,7.234,148.577
C02481=1179.045,247.895,-64.589,-177.321,7.231,148.577
C02482=1179.050,247.646,-64.562,-177.323,7.229,148.577
C02483=1179.054,247.398,-64.535,-177.326,7.226,148.577
C02484=1179.059,247.149,-64.509,-177.329,7.223,148.578
C02485=1179.063,246.901,-64.482,-177.332,7.221,148.578
C02486=1179.068,246.652,-64.455,-177.334,7.218,148.578
C02487=1179.072,246.404,-64.428,-177.337,7.216,148.578
C02488=1179.077,246.155,-64.401,-177.340,7.213,148.578
C02489=1179.081,245.907,-64.374,-177.342,7.211,148.578
C02490=1179.085,245.658,-64.348,-177.345,7.208,148.579
C02491=1179.090,245.410,-64.321,-177.347,7.206,148.579
C02492=1179.094,245.161,-64.295,-177.350,7.203,148.579
C02493=1179.099,244.913,-64.268,-177.353,7.202,148.579
C02494=1179.104,244.664,-64.241,-177.355,7.199,148.579
C02495=1179.108,244.416,-64.215,-177.358,7.196,148.579
C02496=1179.112,244.167,-64.188,-177.361,7.194,148.580
C02497=1179.116,243.918,-64.162,-177.364,7.191,148.580
C02498=1179.121,243.670,-64.135,-177.366,7.189,148.580
C02499=1179.125,243.422,-64.109,-177.369,7.186,148.580
C02500=1179.130,243.173,-64.082,-177.371,7.184,148.580
C02501=1179.134,242.924,-64.056,-177.374,7.181,148.580
C02502=1179.139,242.676,-64.029,-177.377,7.179,148.581
C02503=1179.143,242.427,-64.003,-177.379,7.176,148.581
C02504=1179.147,242.179,-63.976,-177.381,7.174,148.581
C02505=1179.152,241.930,-63.950,-177.385,7.171,148.581
C02506=1179.156,241.681,-63.923,-177.387,7.169,148.581
C02507=1179.160,241.433,-63.897,-177.390,7.166,148.581
C02508=1179.165,241.184,-63.870,-177.392,7.164,148.581
C02509=1179.170,240.936,-63.844,-177.395,7.161,148.582
C02510=1179.175,240.687,-63.818,-177.398,7.160,148.582
C02511=1179.179,240.439,-63.791,-177.400,7.157,148.582
C02512=1179.184,240.190,-63.765,-177.403,7.154,148.582
C02513=1179.187,239.942,-63.739,-177.406,7.152,148.582
C02514=1179.192,239.693,-63.712,-177.409,7.149,148.582
C02515=1179.196,239.445,-63.686,-177.411,7.147,148.583
C02516=1179.201,239.196,-63.660,-177.414,7.144,148.583
C02517=1179.206,238.947,-63.634,-177.416,7.142,148.583
C02518=1179.209,238.698,-63.607,-177.419,7.139,148.583
C02519=1179.215,238.450,-63.581,-177.421,7.137,148.583
C02520=1179.219,238.202,-63.555,-177.425,7.135,148.584
C02521=1179.223,237.953,-63.529,-177.427,7.132,148.584
C02522=1179.228,237.704,-63.503,-177.430,7.129,148.584
C02523=1179.232,237.456,-63.476,-177.432,7.128,148.584
C02524=1179.236,237.207,-63.451,-177.435,7.125,148.584
C02525=1179.241,236.958,-63.423,-177.438,7.123,148.584
C02526=1179.246,236.687,-63.396,-177.440,7.120,148.585
C02527=1179.251,236.416,-63.367,-177.444,7.117,148.585
C02528=1179.256,236.144,-63.338,-177.446,7.115,148.585
C02529=1179.261,235.872,-63.310,-177.449,7.112,148.585
C02530=1179.265,235.624,-63.284,-177.452,7.110,148.585
C02531=1179.270,235.375,-63.258,-177.454,7.108,148.586
C02532=1179.274,235.126,-63.232,-177.457,7.105,148.586
C02533=1179.279,234.878,-63.206,-177.460,7.103,148.586
C02534=1179.283,234.629,-63.180,-177.463,7.100,148.586
C02535=1179.288,234.380,-63.154,-177.465,7.098,148.586
C02536=1179.292,234.132,-63.128,-177.468,7.095,148.586
C02537=1179.297,233.883,-63.102,-177.470,7.093,148.587
C02538=1179.301,233.635,-63.076,-177.473,7.091,148.587
C02539=1179.305,233.386,-63.050,-177.476,7.088,148.587
C02540=1179.310,233.137,-63.024,-177.478,7.086,148.587
C02541=1179.315,232.889,-62.999,-177.481,7.083,148.587
C02542=1179.319,232.640,-62.973,-177.484,7.082,148.588
C02543=1179.323,232.392,-62.947,-177.486,7.079,148.588
C02544=1179.328,232.143,-62.921,-177.489,7.077,148.588
C02545=1179.333,231.894,-62.895,-177.492,7.074,148.588
C02546=1179.337,231.646,-62.870,-177.494,7.072,148.588
C02547=1179.341,231.397,-62.843,-177.497,7.069,148.589
C02548=1179.345,231.149,-62.817,-177.499,7.067,148.589
C02549=1179.350,230.901,-62.792,-177.502,7.065,148.589
C02550=1179.354,230.652,-62.766,-177.505,7.062,148.589
C02551=1179.359,230.403,-62.740,-177.507,7.060,148.589
C02552=1179.363,230.154,-62.714,-177.510,7.057,148.589
C02553=1179.368,229.906,-62.689,-177.513,7.056,148.590
C02554=1179.372,229.657,-62.663,-177.515,7.053,148.590
C02555=1179.377,229.408,-62.637,-177.518,7.051,148.590
C02556=1179.381,229.160,-62.612,-177.521,7.048,148.590
C02557=1179.386,228.911,-62.586,-177.524,7.046,148.591
C02558=1179.390,228.662,-62.561,-177.526,7.044,148.591
C02559=1179.395,228.414,-62.536,-177.529,7.041,148.591
C02560=1179.399,228.165,-62.510,-177.531,7.039,148.591
C02561=1179.403,227.916,-62.484,-177.534,7.037,148.591
C02562=1179.408,227.668,-62.459,-177.537,7.034,148.592
C02563=1179.413,227.419,-62.433,-177.540,7.032,148.592
C02564=1179.417,227.170,-62.407,-177.542,7.030,148.592
C02565=1179.422,226.922,-62.382,-177.545,7.028,148.592
C02566=1179.426,226.673,-62.356,-177.548,7.025,148.593
C02567=1179.430,226.424,-62.331,-177.550,7.023,148.593
C02568=1179.435,226.176,-62.306,-177.553,7.020,148.593
C02569=1179.439,225.927,-62.280,-177.555,7.018,148.593
C02570=1179.444,225.678,-62.254,-177.558,7.017,148.593
C02571=1179.448,225.430,-62.229,-177.561,7.014,148.594
C02572=1179.453,225.181,-62.204,-177.563,7.012,148.594
C02573=1179.458,224.933,-62.178,-177.566,7.009,148.594
C02574=1179.462,224.684,-62.153,-177.569,7.007,148.594
C02575=1179.466,224.435,-62.127,-177.571,7.005,148.594
C02576=1179.471,224.186,-62.102,-177.574,7.002,148.595
C02577=1179.476,223.938,-62.076,-177.576,7.000,148.595
C02578=1179.480,223.689,-62.051,-177.580,6.997,148.595
C02579=1179.485,223.440,-62.026,-177.582,6.996,148.595
C02580=1179.490,223.192,-62.001,-177.584,6.994,148.596
C02581=1179.494,222.943,-61.975,-177.588,6.991,148.596
C02582=1179.498,222.694,-61.950,-177.590,6.989,148.596
C02583=1179.503,222.446,-61.925,-177.593,6.986,148.596
C02584=1179.507,222.197,-61.899,-177.595,6.984,148.596
C02585=1179.512,221.948,-61.875,-177.598,6.982,148.597
C02586=1179.516,221.700,-61.849,-177.601,6.980,148.597
C02587=1179.521,221.451,-61.824,-177.603,6.977,148.597
C02588=1179.526,221.202,-61.798,-177.606,6.976,148.597
C02589=1179.530,220.954,-61.774,-177.609,6.973,148.597
C02590=1179.534,220.705,-61.749,-177.611,6.971,148.598
C02591=1179.539,220.457,-61.723,-177.614,6.968,148.598
C02592=1179.544,220.207,-61.698,-177.617,6.966,148.598
C02593=1179.548,219.959,-61.673,-177.619,6.964,148.599
C02594=1179.552,219.710,-61.648,-177.622,6.961,148.599
C02595=1179.556,219.461,-61.623,-177.625,6.960,148.599
C02596=1179.562,219.213,-61.598,-177.627,6.957,148.599
C02597=1179.566,218.964,-61.573,-177.630,6.955,148.599
C02598=1179.570,218.715,-61.548,-177.633,6.953,148.600
C02599=1179.575,218.467,-61.523,-177.636,6.950,148.600
C02600=1179.580,218.218,-61.498,-177.638,6.948,148.600
C02601=1179.585,217.969,-61.473,-177.641,6.946,148.600
C02602=1179.588,217.721,-61.448,-177.644,6.943,148.601
C02603=1179.593,217.472,-61.423,-177.646,6.942,148.601
C02604=1179.598,217.222,-61.398,-177.649,6.939,148.601
C02605=1179.602,216.975,-61.373,-177.652,6.937,148.601
C02606=1179.606,216.725,-61.348,-177.654,6.935,148.601
C02607=1179.611,216.477,-61.323,-177.657,6.933,148.602
C02608=1179.615,216.228,-61.299,-177.660,6.930,148.602
C02609=1179.620,215.979,-61.274,-177.662,6.928,148.602
C02610=1179.625,215.731,-61.249,-177.665,6.926,148.603
C02611=1179.629,215.482,-61.224,-177.668,6.924,148.603
C02612=1179.634,215.233,-61.199,-177.670,6.922,148.603
C02613=1179.638,214.984,-61.174,-177.673,6.920,148.603
C02614=1179.643,214.736,-61.150,-177.676,6.917,148.603
C02615=1179.647,214.487,-61.125,-177.678,6.915,148.604
C02616=1179.651,214.238,-61.100,-177.681,6.913,148.604
C02617=1179.657,213.990,-61.076,-177.684,6.910,148.604
C02618=1179.661,213.741,-61.050,-177.686,6.909,148.605
C02619=1179.665,213.492,-61.026,-177.689,6.907,148.605
C02620=1179.670,213.244,-61.001,-177.692,6.904,148.605
C02621=1179.674,212.994,-60.977,-177.694,6.902,148.605
C02622=1179.679,212.746,-60.952,-177.697,6.900,148.606
C02623=1179.683,212.497,-60.928,-177.700,6.897,148.606
C02624=1179.688,212.249,-60.902,-177.702,6.895,148.606
C02625=1179.693,212.000,-60.878,-177.705,6.894,148.606
C02626=1179.697,211.751,-60.853,-177.708,6.891,148.606
C02627=1179.702,211.502,-60.829,-177.711,6.889,148.607
C02628=1179.706,211.254,-60.805,-177.713,6.887,148.607
C02629=1179.711,211.004,-60.779,-177.716,6.884,148.607
C02630=1179.716,210.734,-60.753,-177.719,6.882,148.608
C02631=1179.720,210.464,-60.727,-177.722,6.880,148.608
C02632=1179.725,210.193,-60.700,-177.725,6.878,148.608
C02633=1179.730,209.923,-60.673,-177.727,6.875,148.608
C02634=1179.735,209.674,-60.648,-177.730,6.873,148.609
C02635=1179.740,209.426,-60.624,-177.733,6.871,148.609
C02636=1179.744,209.177,-60.599,-177.736,6.869,148.609
C02637=1179.749,208.928,-60.575,-177.738,6.867,148.609
C02638=1179.753,208.679,-60.552,-177.741,6.865,148.610
C02639=1179.758,208.430,-60.527,-177.744,6.862,148.610
C02640=1179.762,208.181,-60.503,-177.746,6.860,148.610
C02641=1179.767,207.932,-60.478,-177.749,6.858,148.611
C02642=1179.772,207.684,-60.454,-177.752,6.856,148.611
C02643=1179.776,207.435,-60.429,-177.754,6.853,148.611
C02644=1179.781,207.186,-60.405,-177.757,6.852,148.611
C02645=1179.785,206.938,-60.381,-177.760,6.850,148.612
C02646=1179.790,206.689,-60.356,-177.762,6.847,148.612
C02647=1179.794,206.440,-60.331,-177.765,6.845,148.612
C02648=1179.798,206.192,-60.307,-177.768,6.843,148.612
C02649=1179.804,205.942,-60.283,-177.770,6.841,148.613
C02650=1179.808,205.694,-60.259,-177.773,6.839,148.613
C02651=1179.812,205.445,-60.235,-177.776,6.837,148.613
C02652=1179.817,205.196,-60.210,-177.778,6.835,148.614
C02653=1179.822,204.948,-60.186,-177.781,6.832,148.614
C02654=1179.826,204.699,-60.163,-177.784,6.830,148.614
C02655=1179.831,204.450,-60.138,-177.786,6.828,148.614
C02656=1179.835,204.201,-60.114,-177.789,6.826,148.614
C02657=1179.840,203.952,-60.090,-177.792,6.824,148.615
C02658=1179.845,203.703,-60.066,-177.795,6.822,148.615
C02659=1179.849,203.455,-60.042,-177.797,6.820,148.615
C02660=1179.854,203.206,-60.018,-177.799,6.818,148.616
C02661=1179.858,202.957,-59.993,-177.803,6.815,148.616
C02662=1179.863,202.708,-59.969,-177.805,6.814,148.616
C02663=1179.867,202.459,-59.945,-177.808,6.812,148.617
C02664=1179.872,202.211,-59.921,-177.810,6.810,148.617
C02665=1179.876,201.962,-59.898,-177.813,6.807,148.617
C02666=1179.881,201.713,-59.874,-177.816,6.805,148.617
C02667=1179.886,201.465,-59.849,-177.818,6.803,148.618
C02668=1179.890,201.215,-59.825,-177.821,6.801,148.618
C02669=1179.894,200.967,-59.801,-177.824,6.799,148.618
C02670=1179.899,200.717,-59.778,-177.827,6.797,148.619
C02671=1179.904,200.469,-59.754,-177.829,6.795,148.619
C02672=1179.908,200.221,-59.730,-177.832,6.793,148.619
C02673=1179.913,199.971,-59.706,-177.835,6.790,148.619
C02674=1179.918,199.723,-59.682,-177.838,6.789,148.620
C02675=1179.923,199.474,-59.658,-177.840,6.786,148.620
C02676=1179.926,199.225,-59.634,-177.842,6.785,148.620
C02677=1179.931,198.976,-59.610,-177.845,6.783,148.620
C02678=1179.935,198.727,-59.586,-177.848,6.780,148.621
C02679=1179.940,198.478,-59.563,-177.850,6.778,148.621
C02680=1179.945,198.230,-59.538,-177.853,6.776,148.621
C02681=1179.950,197.981,-59.515,-177.856,6.775,148.622
C02682=1179.954,197.732,-59.491,-177.859,6.772,148.622
C02683=1179.959,197.483,-59.468,-177.861,6.770,148.622
C02684=1179.963,197.235,-59.443,-177.864,6.768,148.622
C02685=1179.968,196.986,-59.420,-177.867,6.766,148.623
C02686=1179.973,196.737,-59.397,-177.869,6.764,148.623
C02687=1179.977,196.488,-59.373,-177.872,6.762,148.623
C02688=1179.982,196.239,-59.349,-177.875,6.760,148.624
C02689=1179.986,195.991,-59.325,-177.877,6.758,148.624
C02690=1179.990,195.741,-59.302,-177.880,6.756,148.624
C02691=1179.995,195.492,-59.278,-177.883,6.754,148.625
C02692=1180.000,195.244,-59.254,-177.885,6.751,148.625
C02693=1180.004,194.995,-59.231,-177.888,6.750,148.625
C02694=1180.009,194.746,-59.207,-177.891,6.748,148.625
C02695=1180.013,194.497,-59.183,-177.893,6.746,148.626
C02696=1180.018,194.248,-59.160,-177.896,6.744,148.626
C02697=1180.023,193.999,-59.137,-177.899,6.741,148.626
C02698=1180.027,193.750,-59.113,-177.902,6.740,148.627
C02699=1180.032,193.502,-59.089,-177.904,6.738,148.627
C02700=1180.036,193.253,-59.066,-177.907,6.736,148.627
C02701=1180.041,193.004,-59.042,-177.910,6.734,148.628
C02702=1180.046,192.754,-59.019,-177.912,6.732,148.628
C02703=1180.050,192.506,-58.995,-177.915,6.729,148.628
C02704=1180.056,192.258,-58.972,-177.918,6.728,148.628
C02705=1180.060,192.009,-58.949,-177.920,6.726,148.629
C02706=1180.065,191.760,-58.925,-177.923,6.724,148.629
C02707=1180.069,191.511,-58.903,-177.925,6.722,148.629
C02708=1180.073,191.263,-58.878,-177.928,6.719,148.630
C02709=1180.078,191.014,-58.855,-177.931,6.718,148.630
C02710=1180.083,190.764,-58.832,-177.934,6.716,148.630
C02711=1180.087,190.515,-58.808,-177.936,6.714,148.631
C02712=1180.092,190.266,-58.785,-177.939,6.712,148.631
C02713=1180.097,190.017,-58.762,-177.941,6.710,148.631
C02714=1180.102,189.768,-58.738,-177.945,6.707,148.631
C02715=1180.106,189.520,-58.716,-177.947,6.706,148.632
C02716=1180.110,189.271,-58.692,-177.950,6.704,148.632
C02717=1180.115,189.022,-58.669,-177.953,6.702,148.633
C02718=1180.120,188.774,-58.645,-177.955,6.700,148.633
C02719=1180.125,188.525,-58.622,-177.957,6.698,148.633
C02720=1180.129,188.276,-58.599,-177.960,6.696,148.633
C02721=1180.133,188.027,-58.576,-177.963,6.694,148.634
C02722=1180.138,187.778,-58.552,-177.966,6.692,148.634
C02723=1180.143,187.529,-58.529,-177.969,6.690,148.634
C02724=1180.147,187.280,-58.506,-177.971,6.688,148.635
C02725=1180.151,187.031,-58.483,-177.974,6.686,148.635
C02726=1180.157,186.782,-58.460,-177.976,6.685,148.635
C02727=1180.162,186.533,-58.437,-177.979,6.683,148.636
C02728=1180.166,186.284,-58.414,-177.982,6.680,148.636
C02729=1180.170,186.036,-58.391,-177.985,6.678,148.636
C02730=1180.175,185.786,-58.368,-177.987,6.677,148.637
C02731=1180.180,185.537,-58.344,-177.990,6.674,148.637
C02732=1180.184,185.289,-58.322,-177.992,6.673,148.637
C02733=1180.189,185.040,-58.299,-177.995,6.671,148.638
C02734=1180.194,184.771,-58.273,-177.998,6.668,148.638
C02735=1180.199,184.501,-58.249,-178.001,6.667,148.638
C02736=1180.204,184.231,-58.224,-178.004,6.665,148.639
C02737=1180.209,183.962,-58.199,-178.007,6.662,148.639
C02738=1180.213,183.713,-58.176,-178.010,6.660,148.639
C02739=1180.218,183.464,-58.153,-178.012,6.659,148.640
C02740=1180.223,183.215,-58.130,-178.015,6.657,148.640
C02741=1180.227,182.966,-58.107,-178.018,6.655,148.640
C02742=1180.232,182.717,-58.084,-178.020,6.653,148.641
C02743=1180.236,182.468,-58.062,-178.023,6.651,148.641
C02744=1180.241,182.219,-58.038,-178.026,6.648,148.641
C02745=1180.246,181.970,-58.016,-178.028,6.647,148.642
C02746=1180.251,181.722,-57.993,-178.031,6.645,148.642
C02747=1180.255,181.473,-57.970,-178.034,6.643,148.642
C02748=1180.259,181.224,-57.947,-178.036,6.641,148.643
C02749=1180.264,180.974,-57.925,-178.039,6.640,148.643
C02750=1180.269,180.726,-57.902,-178.042,6.638,148.643
C02751=1180.274,180.477,-57.879,-178.044,6.636,148.644
C02752=1180.279,180.228,-57.856,-178.047,6.634,148.644
C02753=1180.283,179.979,-57.833,-178.049,6.632,148.644
C02754=1180.288,179.731,-57.810,-178.052,6.630,148.644
C02755=1180.292,179.481,-57.788,-178.055,6.628,148.645
C02756=1180.297,179.232,-57.765,-178.058,6.626,148.645
C02757=1180.301,178.983,-57.743,-178.061,6.624,148.646
C02758=1180.306,178.735,-57.720,-178.063,6.622,148.646
C02759=1180.310,178.486,-57.697,-178.066,6.621,148.646
C02760=1180.315,178.236,-57.675,-178.069,6.619,148.647
C02761=1180.320,177.988,-57.652,-178.071,6.617,148.647
C02762=1180.325,177.739,-57.629,-178.074,6.615,148.647
C02763=1180.329,177.490,-57.607,-178.076,6.613,148.648
C02764=1180.334,177.241,-57.584,-178.079,6.611,148.648
C02765=1180.338,176.992,-57.562,-178.081,6.610,148.648
C02766=1180.343,176.743,-57.540,-178.084,6.608,148.649
C02767=1180.348,176.494,-57.517,-178.087,6.605,148.649
C02768=1180.352,176.245,-57.495,-178.090,6.603,148.649
C02769=1180.357,175.996,-57.471,-178.093,6.602,148.650
C02770=1180.362,175.747,-57.450,-178.095,6.600,148.650
C02771=1180.367,175.498,-57.426,-178.098,6.598,148.650
C02772=1180.371,175.249,-57.404,-178.101,6.596,148.651
C02773=1180.376,175.000,-57.382,-178.103,6.595,148.651
C02774=1180.380,174.751,-57.359,-178.106,6.593,148.651
C02775=1180.385,174.502,-57.337,-178.109,6.591,148.652
C02776=1180.389,174.254,-57.315,-178.111,6.589,148.652
C02777=1180.394,174.004,-57.292,-178.114,6.587,148.652
C02778=1180.399,173.756,-57.270,-178.116,6.585,148.653
C02779=1180.404,173.507,-57.247,-178.119,6.584,148.653
C02780=1180.408,173.257,-57.225,-178.122,6.582,148.653
C02781=1180.413,173.009,-57.203,-178.124,6.580,148.654
C02782=1180.418,172.760,-57.180,-178.127,6.578,148.654
C02783=1180.423,172.511,-57.158,-178.130,6.576,148.655
C02784=1180.427,172.262,-57.136,-178.132,6.575,148.655
C02785=1180.431,172.013,-57.113,-178.135,6.573,148.655
C02786=1180.436,171.764,-57.091,-178.138,6.571,148.656
C02787=1180.441,171.515,-57.069,-178.141,6.569,148.656
C02788=1180.445,171.266,-57.047,-178.144,6.567,148.656
C02789=1180.450,171.017,-57.024,-178.146,6.565,148.657
C02790=1180.455,170.768,-57.002,-178.149,6.563,148.657
C02791=1180.459,170.519,-56.980,-178.152,6.561,148.657
C02792=1180.464,170.270,-56.959,-178.154,6.560,148.658
C02793=1180.469,170.021,-56.936,-178.157,6.558,148.658
C02794=1180.473,169.772,-56.913,-178.160,6.556,148.659
C02795=1180.478,169.523,-56.892,-178.162,6.554,148.659
C02796=1180.482,169.274,-56.869,-178.165,6.553,148.659
C02797=1180.488,169.025,-56.847,-178.168,6.551,148.660
C02798=1180.492,168.776,-56.825,-178.170,6.549,148.660
C02799=1180.497,168.527,-56.803,-178.173,6.547,148.660
C02800=1180.501,168.278,-56.781,-178.176,6.546,148.661
C02801=1180.506,168.030,-56.759,-178.179,6.544,148.661
C02802=1180.511,167.780,-56.736,-178.181,6.542,148.661
C02803=1180.516,167.531,-56.715,-178.184,6.540,148.662
C02804=1180.520,167.282,-56.693,-178.186,6.538,148.662
C02805=1180.525,167.033,-56.671,-178.189,6.536,148.662
C02806=1180.529,166.784,-56.649,-178.191,6.535,148.663
C02807=1180.534,166.536,-56.627,-178.194,6.533,148.663
C02808=1180.539,166.287,-56.606,-178.197,6.531,148.663
C02809=1180.544,166.037,-56.583,-178.200,6.529,148.664
C02810=1180.549,165.789,-56.561,-178.202,6.527,148.664
C02811=1180.553,165.539,-56.539,-178.205,6.526,148.665
C02812=1180.558,165.291,-56.517,-178.208,6.524,148.665
C02813=1180.562,165.041,-56.495,-178.210,6.522,148.665
C02814=1180.567,164.793,-56.474,-178.213,6.520,148.666
C02815=1180.571,164.543,-56.452,-178.216,6.519,148.666
C02816=1180.576,164.295,-56.430,-178.218,6.517,148.666
C02817=1180.580,164.045,-56.408,-178.221,6.515,148.667
C02818=1180.585,163.797,-56.386,-178.224,6.514,148.667
C02819=1180.590,163.548,-56.365,-178.227,6.512,148.668
C02820=1180.595,163.298,-56.343,-178.229,6.510,148.668
C02821=1180.600,163.049,-56.322,-178.232,6.508,148.668
C02822=1180.604,162.800,-56.300,-178.235,6.507,148.669
C02823=1180.609,162.551,-56.278,-178.238,6.505,148.669
C02824=1180.614,162.303,-56.256,-178.240,6.503,148.670
C02825=1180.618,162.053,-56.234,-178.242,6.502,148.670
C02826=1180.623,161.805,-56.212,-178.245,6.500,148.670
C02827=1180.627,161.555,-56.191,-178.248,6.499,148.671
C02828=1180.632,161.306,-56.169,-178.250,6.497,148.671
C02829=1180.637,161.058,-56.148,-178.253,6.495,148.671
C02830=1180.641,160.808,-56.126,-178.256,6.493,148.672
C02831=1180.646,160.560,-56.104,-178.258,6.491,148.672
C02832=1180.651,160.310,-56.083,-178.261,6.490,148.673
C02833=1180.656,160.061,-56.061,-178.264,6.488,148.673
C02834=1180.661,159.812,-56.039,-178.266,6.486,148.673
C02835=1180.665,159.564,-56.018,-178.269,6.484,148.674
C02836=1180.670,159.314,-55.996,-178.272,6.483,148.674
C02837=1180.675,159.065,-55.975,-178.275,6.481,148.674
C02838=1180.680,158.796,-55.952,-178.277,6.479,148.675
C02839=1180.685,158.527,-55.928,-178.280,6.477,148.675
C02840=1180.690,158.258,-55.905,-178.283,6.476,148.676
C02841=1180.695,157.989,-55.882,-178.286,6.473,148.676
C02842=1180.700,157.740,-55.860,-178.289,6.472,148.677
C02843=1180.705,157.491,-55.839,-178.292,6.470,148.677
C02844=1180.709,157.242,-55.818,-178.294,6.469,148.677
C02845=1180.713,156.993,-55.796,-178.297,6.467,148.678
C02846=1180.719,156.744,-55.775,-178.299,6.465,148.678
C02847=1180.723,156.495,-55.753,-178.302,6.464,148.678
C02848=1180.728,156.245,-55.732,-178.305,6.462,148.679
C02849=1180.733,155.997,-55.710,-178.307,6.460,148.679
C02850=1180.737,155.749,-55.689,-178.310,6.458,148.680
C02851=1180.742,155.499,-55.668,-178.313,6.457,148.680
C02852=1180.746,155.250,-55.646,-178.316,6.455,148.681
C02853=1180.752,155.001,-55.625,-178.318,6.453,148.681
C02854=1180.757,154.752,-55.603,-178.321,6.452,148.681
C02855=1180.760,154.502,-55.583,-178.324,6.450,148.682
C02856=1180.765,154.254,-55.561,-178.327,6.448,148.682
C02857=1180.770,154.004,-55.540,-178.329,6.447,148.682
C02858=1180.775,153.756,-55.518,-178.331,6.445,148.683
C02859=1180.779,153.506,-55.498,-178.334,6.444,148.683
C02860=1180.784,153.258,-55.476,-178.337,6.442,148.684
C02861=1180.789,153.008,-55.455,-178.339,6.440,148.684
C02862=1180.794,152.760,-55.433,-178.342,6.438,148.684
C02863=1180.798,152.511,-55.413,-178.345,6.437,148.685
C02864=1180.803,152.261,-55.392,-178.348,6.435,148.685
C02865=1180.808,152.012,-55.370,-178.351,6.433,148.686
C02866=1180.812,151.763,-55.350,-178.353,6.432,148.686
C02867=1180.817,151.514,-55.328,-178.355,6.431,148.686
C02868=1180.822,151.265,-55.307,-178.358,6.429,148.687
C02869=1180.827,151.015,-55.286,-178.361,6.427,148.687
C02870=1180.831,150.767,-55.265,-178.364,6.425,148.688
C02871=1180.836,150.518,-55.244,-178.366,6.424,148.688
C02872=1180.841,150.268,-55.223,-178.369,6.422,148.688
C02873=1180.846,150.020,-55.201,-178.372,6.420,148.689
C02874=1180.851,149.771,-55.181,-178.375,6.419,148.689
C02875=1180.855,149.521,-55.160,-178.377,6.417,148.690
C02876=1180.860,149.272,-55.139,-178.380,6.416,148.690
C02877=1180.865,149.023,-55.117,-178.382,6.414,148.690
C02878=1180.869,148.774,-55.097,-178.385,6.412,148.691
C02879=1180.874,148.525,-55.076,-178.388,6.411,148.691
C02880=1180.879,148.276,-55.054,-178.390,6.409,148.692
C02881=1180.884,148.027,-55.034,-178.393,6.407,148.692
C02882=1180.888,147.778,-55.012,-178.396,6.405,148.692
C02883=1180.893,147.529,-54.992,-178.399,6.404,148.693
C02884=1180.898,147.279,-54.971,-178.401,6.403,148.693
C02885=1180.902,147.031,-54.950,-178.404,6.401,148.694
C02886=1180.907,146.782,-54.929,-178.406,6.400,148.694
C02887=1180.912,146.532,-54.908,-178.409,6.398,148.695
C02888=1180.917,146.284,-54.888,-178.412,6.396,148.695
C02889=1180.922,146.034,-54.867,-178.414,6.394,148.695
C02890=1180.926,145.785,-54.846,-178.417,6.393,148.696
C02891=1180.931,145.536,-54.825,-178.420,6.392,148.696
C02892=1180.935,145.287,-54.804,-178.422,6.390,148.697
C02893=1180.940,145.038,-54.783,-178.425,6.388,148.697
C02894=1180.945,144.789,-54.763,-178.428,6.387,148.697
C02895=1180.950,144.540,-54.742,-178.430,6.385,148.698
C02896=1180.954,144.291,-54.721,-178.433,6.383,148.698
C02897=1180.959,144.041,-54.700,-178.436,6.381,148.699
C02898=1180.964,143.792,-54.680,-178.438,6.381,148.699
C02899=1180.968,143.543,-54.660,-178.441,6.379,148.700
C02900=1180.973,143.294,-54.639,-178.444,6.377,148.700
C02901=1180.978,143.045,-54.618,-178.447,6.376,148.700
C02902=1180.983,142.796,-54.597,-178.449,6.374,148.701
C02903=1180.987,142.547,-54.577,-178.452,6.372,148.701
C02904=1180.993,142.298,-54.556,-178.454,6.371,148.702
C02905=1180.997,142.049,-54.536,-178.457,6.370,148.702
C02906=1181.002,141.800,-54.515,-178.460,6.368,148.703
C02907=1181.007,141.551,-54.494,-178.463,6.366,148.703
C02908=1181.011,141.302,-54.474,-178.465,6.364,148.703
C02909=1181.016,141.052,-54.453,-178.467,6.363,148.704
C02910=1181.021,140.803,-54.432,-178.470,6.362,148.704
C02911=1181.025,140.554,-54.412,-178.473,6.360,148.705
C02912=1181.030,140.305,-54.391,-178.476,6.359,148.705
C02913=1181.035,140.056,-54.371,-178.479,6.357,148.705
C02914=1181.040,139.807,-54.351,-178.481,6.355,148.706
C02915=1181.045,139.557,-54.330,-178.483,6.354,148.706
C02916=1181.049,139.309,-54.310,-178.486,6.352,148.707
C02917=1181.054,139.060,-54.289,-178.489,6.351,148.707
C02918=1181.059,138.810,-54.268,-178.492,6.349,148.708
C02919=1181.063,138.561,-54.248,-178.495,6.347,148.708
C02920=1181.068,138.312,-54.228,-178.497,6.347,148.708
C02921=1181.073,138.063,-54.207,-178.500,6.345,148.709
C02922=1181.078,137.814,-54.187,-178.503,6.343,148.709
C02923=1181.082,137.565,-54.167,-178.505,6.342,148.710
C02924=1181.086,137.316,-54.146,-178.508,6.340,148.710
C02925=1181.092,137.066,-54.126,-178.510,6.339,148.711
C02926=1181.097,136.818,-54.106,-178.513,6.337,148.711
C02927=1181.101,136.569,-54.086,-178.516,6.335,148.711
C02928=1181.107,136.319,-54.065,-178.519,6.334,148.712
C02929=1181.111,136.070,-54.045,-178.522,6.332,148.712
C02930=1181.116,135.821,-54.025,-178.524,6.331,148.713
C02931=1181.120,135.572,-54.004,-178.526,6.330,148.713
C02932=1181.125,135.322,-53.985,-178.529,6.328,148.714
C02933=1181.130,135.073,-53.964,-178.532,6.326,148.714
C02934=1181.135,134.824,-53.943,-178.534,6.325,148.715
C02935=1181.139,134.575,-53.924,-178.537,6.324,148.715
C02936=1181.144,134.326,-53.904,-178.540,6.322,148.715
C02937=1181.149,134.077,-53.883,-178.542,6.320,148.716
C02938=1181.154,133.827,-53.863,-178.546,6.319,148.716
C02939=1181.159,133.579,-53.843,-178.548,6.318,148.717
C02940=1181.163,133.330,-53.822,-178.550,6.316,148.717
C02941=1181.168,133.080,-53.803,-178.553,6.314,148.718
C02942=1181.173,132.812,-53.780,-178.556,6.313,148.718
C02943=1181.178,132.543,-53.759,-178.559,6.311,148.719
C02944=1181.184,132.274,-53.737,-178.562,6.310,148.719
C02945=1181.188,132.006,-53.716,-178.565,6.308,148.720
C02946=1181.193,131.756,-53.696,-178.568,6.306,148.720
C02947=1181.198,131.508,-53.676,-178.570,6.305,148.720
C02948=1181.203,131.259,-53.656,-178.573,6.304,148.721
C02949=1181.208,131.009,-53.635,-178.576,6.302,148.721
C02950=1181.213,130.760,-53.616,-178.578,6.301,148.722
C02951=1181.217,130.511,-53.595,-178.580,6.300,148.722
C02952=1181.223,130.262,-53.576,-178.583,6.298,148.723
C02953=1181.227,130.013,-53.556,-178.586,6.296,148.723
C02954=1181.232,129.763,-53.536,-178.589,6.295,148.724
C02955=1181.236,129.515,-53.516,-178.591,6.294,148.724
C02956=1181.241,129.265,-53.496,-178.594,6.292,148.724
C02957=1181.246,129.016,-53.477,-178.597,6.291,148.725
C02958=1181.251,128.767,-53.456,-178.600,6.289,148.725
C02959=1181.255,128.518,-53.437,-178.602,6.288,148.726
C02960=1181.260,128.269,-53.416,-178.604,6.286,148.726
C02961=1181.265,128.020,-53.397,-178.608,6.285,148.727
C02962=1181.270,127.770,-53.377,-178.610,6.283,148.727
C02963=1181.274,127.521,-53.357,-178.612,6.282,148.728
C02964=1181.279,127.272,-53.337,-178.615,6.280,148.728
C02965=1181.285,127.023,-53.318,-178.618,6.279,148.729
C02966=1181.289,126.774,-53.298,-178.621,6.278,148.729
C02967=1181.294,126.524,-53.278,-178.623,6.276,148.729
C02968=1181.298,126.275,-53.258,-178.626,6.275,148.730
C02969=1181.303,126.026,-53.238,-178.629,6.273,148.730
C02970=1181.308,125.777,-53.219,-178.631,6.272,148.731
C02971=1181.313,125.527,-53.199,-178.634,6.271,148.731
C02972=1181.317,125.278,-53.179,-178.637,6.269,148.732
C02973=1181.323,125.030,-53.159,-178.639,6.268,148.732
C02974=1181.328,124.780,-53.140,-178.642,6.266,148.733
C02975=1181.332,124.530,-53.120,-178.645,6.265,148.733
C02976=1181.337,124.282,-53.101,-178.647,6.263,148.733
C02977=1181.341,124.033,-53.081,-178.650,6.262,148.734
C02978=1181.346,123.783,-53.061,-178.653,6.261,148.734
C02979=1181.351,123.534,-53.042,-178.655,6.259,148.735
C02980=1181.356,123.285,-53.022,-178.658,6.258,148.735
C02981=1181.361,123.036,-53.002,-178.661,6.257,148.736
C02982=1181.366,122.787,-52.983,-178.663,6.255,148.736
C02983=1181.371,122.537,-52.963,-178.666,6.253,148.737
C02984=1181.375,122.288,-52.944,-178.669,6.253,148.737
C02985=1181.380,122.039,-52.925,-178.671,6.251,148.738
C02986=1181.385,121.790,-52.905,-178.674,6.249,148.738
C02987=1181.389,121.540,-52.885,-178.676,6.248,148.738
C02988=1181.395,121.292,-52.865,-178.679,6.247,148.739
C02989=1181.399,121.042,-52.846,-178.682,6.245,148.739
C02990=1181.403,120.793,-52.827,-178.684,6.244,148.740
C02991=1181.409,120.544,-52.807,-178.687,6.243,148.741
C02992=1181.413,120.295,-52.788,-178.690,6.241,148.741
C02993=1181.419,120.046,-52.768,-178.692,6.240,148.741
C02994=1181.423,119.796,-52.749,-178.695,6.238,148.742
C02995=1181.427,119.547,-52.730,-178.698,6.237,148.742
C02996=1181.433,119.298,-52.710,-178.700,6.236,148.743
C02997=1181.438,119.049,-52.691,-178.703,6.234,148.743
C02998=1181.443,118.800,-52.671,-178.706,6.233,148.744
C02999=1181.447,118.550,-52.652,-178.708,6.232,148.744
C03000=1181.452,118.301,-52.633,-178.711,6.230,148.745
C03001=1181.457,118.052,-52.613,-178.714,6.229,148.745
C03002=1181.462,117.802,-52.594,-178.716,6.228,148.746
C03003=1181.466,117.554,-52.575,-178.719,6.226,148.746
C03004=1181.471,117.304,-52.555,-178.722,6.224,148.746
C03005=1181.476,117.055,-52.536,-178.724,6.224,148.747
C03006=1181.480,116.806,-52.517,-178.727,6.222,148.747
C03007=1181.485,116.557,-52.497,-178.730,6.220,148.748
C03008=1181.491,116.307,-52.479,-178.732,6.220,148.749
C03009=1181.495,116.058,-52.460,-178.735,6.218,148.749
C03010=1181.500,115.809,-52.441,-178.738,6.216,148.749
C03011=1181.505,115.559,-52.421,-178.740,6.216,148.750
C03012=1181.509,115.311,-52.402,-178.743,6.214,148.750
C03013=1181.514,115.061,-52.383,-178.746,6.212,148.751
C03014=1181.520,114.812,-52.363,-178.748,6.212,148.751
C03015=1181.524,114.563,-52.345,-178.751,6.210,148.752
C03016=1181.529,114.314,-52.326,-178.754,6.208,148.752
C03017=1181.534,114.064,-52.306,-178.756,6.208,148.753
C03018=1181.539,113.816,-52.287,-178.759,6.206,148.753
C03019=1181.543,113.566,-52.268,-178.761,6.205,148.754
C03020=1181.548,113.317,-52.250,-178.764,6.204,148.754
C03021=1181.553,113.067,-52.230,-178.767,6.202,148.755
C03022=1181.558,112.818,-52.211,-178.769,6.201,148.755
C03023=1181.562,112.569,-52.192,-178.772,6.200,148.756
C03024=1181.568,112.320,-52.173,-178.775,6.198,148.756
C03025=1181.572,112.070,-52.154,-178.777,6.197,148.757
C03026=1181.577,111.822,-52.135,-178.780,6.196,148.757
C03027=1181.581,111.572,-52.116,-178.783,6.194,148.758
C03028=1181.587,111.323,-52.097,-178.785,6.193,148.758
C03029=1181.592,111.074,-52.078,-178.788,6.192,148.759
C03030=1181.596,110.825,-52.059,-178.791,6.191,148.759
C03031=1181.602,110.575,-52.040,-178.793,6.189,148.759
C03032=1181.606,110.326,-52.021,-178.797,6.188,148.760
C03033=1181.611,110.077,-52.002,-178.799,6.187,148.760
C03034=1181.616,109.827,-51.983,-178.801,6.185,148.761
C03035=1181.621,109.578,-51.964,-178.804,6.184,148.762
C03036=1181.625,109.329,-51.945,-178.807,6.183,148.762
C03037=1181.631,109.080,-51.927,-178.809,6.181,148.762
C03038=1181.635,108.831,-51.908,-178.812,6.180,148.763
C03039=1181.640,108.581,-51.889,-178.815,6.179,148.763
C03040=1181.645,108.332,-51.870,-178.817,6.177,148.764
C03041=1181.649,108.083,-51.851,-178.820,6.176,148.764
C03042=1181.655,107.834,-51.833,-178.823,6.175,148.765
C03043=1181.659,107.585,-51.814,-178.825,6.174,148.765
C03044=1181.664,107.335,-51.795,-178.828,6.172,148.766
C03045=1181.669,107.086,-51.776,-178.831,6.170,148.766
C03046=1181.675,106.818,-51.756,-178.833,6.170,148.767
C03047=1181.679,106.549,-51.736,-178.836,6.168,148.767
C03048=1181.685,106.281,-51.716,-178.839,6.167,148.768
C03049=1181.690,106.012,-51.696,-178.842,6.165,148.768
C03050=1181.694,105.763,-51.677,-178.845,6.165,148.769
C03051=1181.699,105.514,-51.659,-178.847,6.163,148.769
C03052=1181.705,105.265,-51.639,-178.849,6.162,148.770
C03053=1181.709,105.015,-51.621,-178.853,6.161,148.770
C03054=1181.714,104.766,-51.602,-178.855,6.159,148.771
C03055=1181.719,104.517,-51.584,-178.858,6.158,148.772
C03056=1181.724,104.267,-51.565,-178.861,6.156,148.772
C03057=1181.728,104.019,-51.547,-178.863,6.156,148.772
C03058=1181.734,103.769,-51.528,-178.866,6.154,148.773
C03059=1181.738,103.520,-51.509,-178.868,6.153,148.773
C03060=1181.743,103.271,-51.491,-178.871,6.152,148.774
C03061=1181.748,103.021,-51.473,-178.874,6.150,148.774
C03062=1181.752,102.772,-51.453,-178.876,6.149,148.775
C03063=1181.757,102.523,-51.435,-178.879,6.148,148.775
C03064=1181.763,102.273,-51.417,-178.882,6.147,148.776
C03065=1181.767,102.024,-51.398,-178.884,6.145,148.776
C03066=1181.772,101.775,-51.380,-178.887,6.145,148.777
C03067=1181.778,101.525,-51.361,-178.890,6.143,148.777
C03068=1181.782,101.277,-51.343,-178.893,6.142,148.778
C03069=1181.786,101.027,-51.324,-178.895,6.141,148.778
C03070=1181.791,100.778,-51.306,-178.898,6.139,148.779
C03071=1181.797,100.528,-51.288,-178.900,6.138,148.779
C03072=1181.801,100.279,-51.269,-178.903,6.137,148.780
C03073=1181.806,100.030,-51.251,-178.906,6.136,148.781
C03074=1181.811,99.781,-51.233,-178.908,6.134,148.781
C03075=1181.816,99.531,-51.215,-178.910,6.134,148.781
C03076=1181.821,99.282,-51.195,-178.914,6.132,148.782
C03077=1181.825,99.033,-51.177,-178.916,6.131,148.782
C03078=1181.830,98.784,-51.159,-178.919,6.130,148.783
C03079=1181.835,98.534,-51.141,-178.922,6.128,148.783
C03080=1181.840,98.285,-51.123,-178.924,6.127,148.784
C03081=1181.845,98.036,-51.103,-178.927,6.126,148.785
C03082=1181.850,97.786,-51.085,-178.929,6.125,148.785
C03083=1181.855,97.537,-51.067,-178.932,6.124,148.786
C03084=1181.860,97.288,-51.050,-178.934,6.123,148.786
C03085=1181.864,97.038,-51.031,-178.937,6.121,148.786
C03086=1181.869,96.789,-51.013,-178.940,6.120,148.787
C03087=1181.875,96.540,-50.995,-178.943,6.119,148.787
C03088=1181.879,96.291,-50.976,-178.945,6.118,148.788
C03089=1181.884,96.042,-50.958,-178.948,6.116,148.789
C03090=1181.889,95.793,-50.940,-178.950,6.116,148.789
C03091=1181.893,95.543,-50.922,-178.953,6.114,148.790
C03092=1181.898,95.294,-50.904,-178.955,6.113,148.790
C03093=1181.903,95.044,-50.886,-178.959,6.112,148.791
C03094=1181.908,94.795,-50.868,-178.961,6.111,148.791
C03095=1181.913,94.546,-50.850,-178.964,6.110,148.792
C03096=1181.919,94.297,-50.831,-178.966,6.109,148.792
C03097=1181.923,94.047,-50.813,-178.969,6.107,148.793
C03098=1181.928,93.797,-50.795,-178.971,6.106,148.793
C03099=1181.933,93.548,-50.777,-178.974,6.105,148.794
C03100=1181.938,93.299,-50.759,-178.977,6.104,148.794
C03101=1181.943,93.050,-50.741,-178.979,6.102,148.795
C03102=1181.947,92.801,-50.723,-178.983,6.101,148.795
C03103=1181.952,92.552,-50.705,-178.985,6.100,148.796
C03104=1181.957,92.302,-50.687,-178.988,6.099,148.796
C03105=1181.962,92.053,-50.669,-178.990,6.098,148.797
C03106=1181.966,91.803,-50.651,-178.992,6.097,148.797
C03107=1181.971,91.554,-50.633,-178.995,6.096,148.798
C03108=1181.977,91.304,-50.615,-178.998,6.095,148.798
C03109=1181.982,91.055,-50.597,-179.001,6.093,148.799
C03110=1181.986,90.806,-50.579,-179.003,6.092,148.799
C03111=1181.991,90.557,-50.561,-179.006,6.091,148.800
C03112=1181.996,90.308,-50.543,-179.008,6.090,148.800
C03113=1182.001,90.058,-50.525,-179.011,6.089,148.801
C03114=1182.005,89.809,-50.507,-179.014,6.088,148.802
C03115=1182.010,89.559,-50.489,-179.016,6.086,148.802
C03116=1182.016,89.310,-50.472,-179.019,6.086,148.803
C03117=1182.021,89.061,-50.454,-179.022,6.084,148.803
C03118=1182.025,88.812,-50.436,-179.024,6.083,148.804
C03119=1182.030,88.562,-50.419,-179.027,6.082,148.804
C03120=1182.035,88.313,-50.401,-179.030,6.081,148.805
C03121=1182.040,88.063,-50.383,-179.032,6.079,148.805
C03122=1182.045,87.814,-50.365,-179.035,6.079,148.806
C03123=1182.050,87.565,-50.347,-179.038,6.077,148.806
C03124=1182.054,87.316,-50.329,-179.040,6.077,148.807
C03125=1182.060,87.066,-50.312,-179.043,6.075,148.807
C03126=1182.065,86.817,-50.294,-179.045,6.074,148.808
C03127=1182.070,86.568,-50.276,-179.048,6.073,148.808
C03128=1182.074,86.319,-50.259,-179.050,6.072,148.809
C03129=1182.079,86.069,-50.241,-179.053,6.071,148.809
C03130=1182.084,85.820,-50.223,-179.056,6.069,148.810
C03131=1182.089,85.571,-50.206,-179.058,6.069,148.810
C03132=1182.094,85.321,-50.188,-179.061,6.067,148.811
C03133=1182.099,85.072,-50.170,-179.064,6.067,148.812
C03134=1182.103,84.823,-50.153,-179.066,6.065,148.812
C03135=1182.108,84.573,-50.136,-179.069,6.064,148.813
C03136=1182.113,84.324,-50.118,-179.072,6.063,148.813
C03137=1182.118,84.074,-50.100,-179.074,6.062,148.814
C03138=1182.123,83.825,-50.082,-179.077,6.060,148.814
C03139=1182.127,83.576,-50.065,-179.080,6.060,148.815
C03140=1182.133,83.326,-50.048,-179.082,6.059,148.815
C03141=1182.138,83.077,-50.030,-179.085,6.058,148.816
C03142=1182.143,82.827,-50.012,-179.087,6.057,148.816
C03143=1182.148,82.578,-49.995,-179.090,6.055,148.817
C03144=1182.152,82.329,-49.977,-179.093,6.054,148.817
C03145=1182.157,82.080,-49.960,-179.095,6.053,148.818
C03146=1182.162,81.830,-49.942,-179.098,6.052,148.818
C03147=1182.167,81.581,-49.925,-179.100,6.051,148.819
C03148=1182.171,81.332,-49.907,-179.103,6.050,148.820
C03149=1182.177,81.082,-49.890,-179.105,6.049,148.820
C03150=1182.182,80.814,-49.871,-179.109,6.048,148.821
C03151=1182.188,80.546,-49.852,-179.112,6.046,148.821
C03152=1182.192,80.277,-49.834,-179.114,6.045,148.822
C03153=1182.197,80.009,-49.815,-179.117,6.044,148.822
C03154=1182.203,79.760,-49.798,-179.120,6.044,148.823
C03155=1182.208,79.510,-49.780,-179.123,6.042,148.823
C03156=1182.213,79.261,-49.763,-179.125,6.041,148.824
C03157=1182.218,79.011,-49.746,-179.127,6.040,148.824
C03158=1182.223,78.762,-49.728,-179.131,6.039,148.825
C03159=1182.227,78.512,-49.711,-179.133,6.038,148.826
C03160=1182.232,78.263,-49.693,-179.136,6.037,148.826
C03161=1182.237,78.014,-49.677,-179.138,6.036,148.827
C03162=1182.242,77.764,-49.659,-179.141,6.035,148.827
C03163=1182.247,77.516,-49.642,-179.143,6.034,148.828
C03164=1182.252,77.266,-49.625,-179.146,6.033,148.828
C03165=1182.257,77.017,-49.607,-179.149,6.031,148.829
C03166=1182.262,76.767,-49.590,-179.151,6.031,148.829
C03167=1182.266,76.518,-49.573,-179.154,6.029,148.830
C03168=1182.271,76.268,-49.555,-179.157,6.029,148.831
C03169=1182.276,76.019,-49.539,-179.159,6.028,148.831
C03170=1182.282,75.770,-49.522,-179.162,6.026,148.832
C03171=1182.287,75.521,-49.504,-179.164,6.025,148.832
C03172=1182.291,75.271,-49.487,-179.167,6.025,148.833
C03173=1182.296,75.021,-49.470,-179.170,6.023,148.833
C03174=1182.301,74.772,-49.453,-179.172,6.023,148.834
C03175=1182.306,74.523,-49.435,-179.175,6.021,148.834
C03176=1182.311,74.274,-49.419,-179.178,6.020,148.835
C03177=1182.316,74.024,-49.401,-179.180,6.020,148.835
C03178=1182.320,73.775,-49.385,-179.183,6.018,148.836
C03179=1182.325,73.526,-49.367,-179.185,6.017,148.836
C03180=1182.330,73.276,-49.350,-179.188,6.016,148.837
C03181=1182.336,73.027,-49.333,-179.190,6.015,148.837
C03182=1182.340,72.777,-49.317,-179.193,6.015,148.838
C03183=1182.345,72.528,-49.299,-179.196,6.013,148.839
C03184=1182.350,72.279,-49.282,-179.198,6.012,148.839
C03185=1182.355,72.030,-49.265,-179.201,6.012,148.840
C03186=1182.360,71.780,-49.248,-179.204,6.010,148.840
C03187=1182.365,71.530,-49.231,-179.206,6.010,148.841
C03188=1182.370,71.281,-49.214,-179.209,6.008,148.841
C03189=1182.375,71.032,-49.198,-179.212,6.007,148.842
C03190=1182.380,70.782,-49.181,-179.214,6.006,148.842
C03191=1182.385,70.533,-49.164,-179.217,6.005,148.843
C03192=1182.389,70.284,-49.146,-179.219,6.004,148.844
C03193=1182.395,70.035,-49.129,-179.222,6.004,148.844
C03194=1182.400,69.785,-49.113,-179.225,6.002,148.845
C03195=1182.404,69.536,-49.096,-179.227,6.001,148.845
C03196=1182.409,69.286,-49.079,-179.229,6.000,148.846
C03197=1182.414,69.037,-49.062,-179.233,5.999,148.846
C03198=1182.420,68.787,-49.045,-179.235,5.998,148.847
C03199=1182.424,68.538,-49.028,-179.237,5.998,148.847
C03200=1182.429,68.288,-49.012,-179.241,5.996,148.848
C03201=1182.434,68.039,-48.995,-179.243,5.995,148.849
C03202=1182.439,67.790,-48.978,-179.246,5.994,148.849
C03203=1182.444,67.540,-48.961,-179.248,5.993,148.850
C03204=1182.449,67.291,-48.945,-179.251,5.993,148.850
C03205=1182.454,67.042,-48.928,-179.253,5.991,148.851
C03206=1182.459,66.792,-48.911,-179.256,5.991,148.851
C03207=1182.464,66.543,-48.894,-179.258,5.990,148.852
C03208=1182.468,66.294,-48.878,-179.261,5.988,148.853
C03209=1182.474,66.044,-48.861,-179.264,5.987,148.853
C03210=1182.479,65.795,-48.844,-179.266,5.987,148.854
C03211=1182.483,65.546,-48.828,-179.269,5.986,148.854
C03212=1182.488,65.296,-48.810,-179.272,5.985,148.855
C03213=1182.493,65.047,-48.794,-179.274,5.984,148.855
C03214=1182.498,64.797,-48.778,-179.277,5.982,148.856
C03215=1182.503,64.547,-48.761,-179.280,5.982,148.856
C03216=1182.509,64.298,-48.744,-179.282,5.981,148.857
C03217=1182.513,64.049,-48.728,-179.285,5.980,148.858
C03218=1182.517,63.799,-48.711,-179.287,5.979,148.858
C03219=1182.523,63.551,-48.695,-179.290,5.978,148.859
C03220=1182.528,63.301,-48.678,-179.292,5.978,148.859
C03221=1182.533,63.051,-48.662,-179.295,5.976,148.860
C03222=1182.538,62.802,-48.645,-179.298,5.975,148.860
C03223=1182.542,62.552,-48.629,-179.300,5.975,148.861
C03224=1182.548,62.303,-48.612,-179.303,5.973,148.862
C03225=1182.552,62.054,-48.595,-179.305,5.972,148.862
C03226=1182.557,61.804,-48.578,-179.308,5.972,148.863
C03227=1182.562,61.555,-48.563,-179.311,5.971,148.863
C03228=1182.568,61.305,-48.546,-179.313,5.970,148.864
C03229=1182.573,61.056,-48.529,-179.316,5.969,148.864
C03230=1182.577,60.807,-48.513,-179.319,5.967,148.865
C03231=1182.582,60.557,-48.497,-179.321,5.967,148.865
C03232=1182.587,60.308,-48.480,-179.323,5.966,148.866
C03233=1182.592,60.058,-48.463,-179.326,5.965,148.867
C03234=1182.598,59.809,-48.447,-179.329,5.964,148.867
C03235=1182.602,59.559,-48.431,-179.331,5.963,148.868
C03236=1182.607,59.310,-48.414,-179.334,5.963,148.868
C03237=1182.612,59.061,-48.398,-179.337,5.961,148.869
C03238=1182.617,58.812,-48.382,-179.339,5.961,148.869
C03239=1182.621,58.562,-48.366,-179.342,5.960,148.870
C03240=1182.627,58.312,-48.348,-179.345,5.958,148.871
C03241=1182.632,58.063,-48.333,-179.347,5.958,148.871
C03242=1182.637,57.813,-48.316,-179.350,5.957,148.872
C03243=1182.642,57.564,-48.300,-179.352,5.956,148.872
C03244=1182.646,57.315,-48.284,-179.355,5.955,148.873
C03245=1182.651,57.066,-48.267,-179.358,5.954,148.873
C03246=1182.656,56.816,-48.252,-179.360,5.953,148.874
C03247=1182.661,56.567,-48.235,-179.363,5.952,148.874
C03248=1182.666,56.317,-48.219,-179.366,5.951,148.875
C03249=1182.672,56.068,-48.202,-179.368,5.951,148.876
C03250=1182.676,55.818,-48.186,-179.370,5.950,148.876
C03251=1182.682,55.569,-48.170,-179.373,5.948,148.877
C03252=1182.686,55.319,-48.153,-179.376,5.948,148.877
C03253=1182.692,55.070,-48.138,-179.378,5.947,148.878
C03254=1182.697,54.802,-48.120,-179.381,5.946,148.878
C03255=1182.702,54.533,-48.103,-179.384,5.945,148.879
C03256=1182.707,54.264,-48.086,-179.386,5.945,148.880
C03257=1182.713,53.996,-48.069,-179.390,5.943,148.880
C03258=1182.717,53.746,-48.052,-179.392,5.942,148.881
C03259=1182.723,53.497,-48.036,-179.394,5.942,148.882
C03260=1182.727,53.248,-48.020,-179.398,5.940,148.882
C03261=1182.733,52.998,-48.004,-179.400,5.940,148.883
C03262=1182.737,52.749,-47.988,-179.402,5.939,148.883
C03263=1182.743,52.499,-47.972,-179.404,5.938,148.884
C03264=1182.748,52.250,-47.956,-179.408,5.937,148.884
C03265=1182.752,52.000,-47.940,-179.410,5.936,148.885
C03266=1182.758,51.751,-47.924,-179.412,5.935,148.886
C03267=1182.762,51.501,-47.907,-179.415,5.935,148.886
C03268=1182.768,51.252,-47.892,-179.418,5.933,148.887
C03269=1182.772,51.003,-47.875,-179.420,5.933,148.887
C03270=1182.778,50.753,-47.860,-179.423,5.932,148.888
C03271=1182.782,50.503,-47.844,-179.425,5.931,148.888
C03272=1182.787,50.254,-47.827,-179.429,5.930,148.889
C03273=1182.793,50.005,-47.812,-179.431,5.929,148.890
C03274=1182.797,49.755,-47.796,-179.433,5.929,148.890
C03275=1182.802,49.506,-47.780,-179.436,5.928,148.891
C03276=1182.807,49.256,-47.764,-179.439,5.926,148.891
C03277=1182.812,49.007,-47.749,-179.441,5.926,148.892
C03278=1182.817,48.758,-47.732,-179.443,5.925,148.892
C03279=1182.822,48.508,-47.716,-179.446,5.925,148.893
C03280=1182.827,48.259,-47.701,-179.449,5.923,148.894
C03281=1182.832,48.010,-47.684,-179.451,5.922,148.894
C03282=1182.837,47.760,-47.668,-179.454,5.922,148.895
C03283=1182.842,47.511,-47.653,-179.457,5.921,148.896
C03284=1182.847,47.260,-47.637,-179.459,5.920,148.896
C03285=1182.852,47.012,-47.621,-179.462,5.919,148.897
C03286=1182.857,46.762,-47.606,-179.464,5.918,148.897
C03287=1182.862,46.512,-47.590,-179.467,5.918,148.898
C03288=1182.867,46.263,-47.574,-179.470,5.917,148.898
C03289=1182.872,46.014,-47.558,-179.472,5.916,148.899
C03290=1182.876,45.764,-47.542,-179.475,5.915,148.900
C03291=1182.882,45.515,-47.527,-179.477,5.914,148.900
C03292=1182.887,45.265,-47.511,-179.480,5.914,148.901
C03293=1182.892,45.015,-47.495,-179.482,5.913,148.901
C03294=1182.896,44.767,-47.480,-179.485,5.911,148.902
C03295=1182.902,44.517,-47.464,-179.488,5.911,148.902
C03296=1182.907,44.267,-47.448,-179.490,5.910,148.903
C03297=1182.912,44.018,-47.432,-179.493,5.910,148.904
C03298=1182.917,43.769,-47.417,-179.495,5.909,148.904
C03299=1182.922,43.519,-47.402,-179.498,5.907,148.905
C03300=1182.927,43.269,-47.386,-179.501,5.907,148.905
C03301=1182.932,43.020,-47.370,-179.503,5.906,148.906
C03302=1182.936,42.771,-47.355,-179.505,5.905,148.906
C03303=1182.941,42.521,-47.339,-179.508,5.905,148.907
C03304=1182.947,42.272,-47.323,-179.511,5.904,148.908
C03305=1182.952,42.023,-47.307,-179.513,5.903,148.908
C03306=1182.957,41.773,-47.292,-179.516,5.902,148.909
C03307=1182.961,41.523,-47.276,-179.518,5.901,148.909
C03308=1182.967,41.274,-47.261,-179.521,5.901,148.910
C03309=1182.972,41.025,-47.246,-179.524,5.900,148.911
C03310=1182.977,40.775,-47.230,-179.526,5.899,148.911
C03311=1182.982,40.525,-47.214,-179.529,5.898,148.912
C03312=1182.987,40.276,-47.199,-179.531,5.898,148.913
C03313=1182.992,40.027,-47.184,-179.534,5.897,148.913
C03314=1182.997,39.777,-47.168,-179.536,5.896,148.914
C03315=1183.002,39.527,-47.152,-179.539,5.895,148.914
C03316=1183.007,39.278,-47.137,-179.542,5.894,148.915
C03317=1183.012,39.029,-47.122,-179.544,5.894,148.915
C03318=1183.017,38.779,-47.106,-179.546,5.893,148.916
C03319=1183.022,38.530,-47.091,-179.549,5.892,148.917
C03320=1183.027,38.280,-47.075,-179.552,5.891,148.917
C03321=1183.031,38.031,-47.060,-179.554,5.890,148.918
C03322=1183.037,37.782,-47.045,-179.557,5.890,148.918
C03323=1183.042,37.532,-47.030,-179.560,5.889,148.919
C03324=1183.047,37.283,-47.015,-179.562,5.888,148.919
C03325=1183.052,37.033,-46.999,-179.565,5.888,148.920
C03326=1183.057,36.783,-46.984,-179.568,5.886,148.921
C03327=1183.062,36.534,-46.968,-179.570,5.885,148.921
C03328=1183.067,36.285,-46.953,-179.573,5.885,148.922
C03329=1183.072,36.036,-46.938,-179.575,5.884,148.923
C03330=1183.077,35.785,-46.922,-179.577,5.884,148.923
C03331=1183.082,35.536,-46.907,-179.580,5.883,148.924
C03332=1183.087,35.286,-46.892,-179.583,5.883,148.924
C03333=1183.092,35.037,-46.877,-179.585,5.881,148.925
C03334=1183.097,34.788,-46.861,-179.588,5.880,148.926
C03335=1183.103,34.538,-46.846,-179.590,5.880,148.926
C03336=1183.108,34.289,-46.831,-179.593,5.879,148.927
C03337=1183.112,34.039,-46.815,-179.595,5.879,148.927
C03338=1183.117,33.790,-46.800,-179.598,5.878,148.928
C03339=1183.122,33.540,-46.785,-179.601,5.876,148.928
C03340=1183.127,33.291,-46.770,-179.604,5.876,148.929
C03341=1183.133,33.041,-46.755,-179.606,5.875,148.930
C03342=1183.137,32.792,-46.740,-179.608,5.874,148.930
C03343=1183.143,32.543,-46.724,-179.611,5.874,148.931
C03344=1183.148,32.293,-46.710,-179.613,5.873,148.931
C03345=1183.152,32.043,-46.694,-179.616,5.873,148.932
C03346=1183.157,31.794,-46.679,-179.619,5.871,148.933
C03347=1183.162,31.545,-46.664,-179.621,5.870,148.933
C03348=1183.167,31.294,-46.649,-179.624,5.870,148.934
C03349=1183.172,31.045,-46.634,-179.626,5.869,148.935
C03350=1183.177,30.796,-46.619,-179.629,5.869,148.935
C03351=1183.182,30.546,-46.604,-179.631,5.868,148.936
C03352=1183.188,30.297,-46.589,-179.634,5.868,148.936
C03353=1183.192,30.048,-46.574,-179.636,5.867,148.937
C03354=1183.198,29.798,-46.559,-179.639,5.865,148.937
C03355=1183.203,29.549,-46.544,-179.642,5.865,148.938
C03356=1183.207,29.299,-46.529,-179.644,5.864,148.939
C03357=1183.213,29.049,-46.514,-179.647,5.864,148.939
C03358=1183.218,28.780,-46.498,-179.649,5.863,148.940
C03359=1183.224,28.511,-46.482,-179.652,5.863,148.941
C03360=1183.228,28.243,-46.465,-179.655,5.861,148.941
C03361=1183.234,27.974,-46.449,-179.657,5.860,148.942
C03362=1183.239,27.724,-46.435,-179.660,5.860,148.942
C03363=1183.244,27.475,-46.420,-179.663,5.859,148.943
C03364=1183.249,27.225,-46.404,-179.665,5.859,148.944
C03365=1183.254,26.976,-46.390,-179.668,5.858,148.944
C03366=1183.259,26.727,-46.375,-179.671,5.857,148.945
C03367=1183.265,26.477,-46.360,-179.673,5.856,148.945
C03368=1183.269,26.228,-46.345,-179.676,5.855,148.946
C03369=1183.274,25.978,-46.331,-179.678,5.855,148.947
C03370=1183.279,25.728,-46.315,-179.681,5.854,148.947
C03371=1183.284,25.479,-46.301,-179.683,5.853,148.948
C03372=1183.289,25.230,-46.286,-179.686,5.853,148.949
C03373=1183.295,24.980,-46.271,-179.688,5.853,148.949
C03374=1183.299,24.731,-46.256,-179.690,5.852,148.950
C03375=1183.304,24.481,-46.242,-179.693,5.851,148.950
C03376=1183.310,24.231,-46.227,-179.696,5.850,148.951
C03377=1183.315,23.982,-46.212,-179.699,5.849,148.951
C03378=1183.320,23.732,-46.198,-179.701,5.848,148.952
C03379=1183.324,23.483,-46.183,-179.704,5.848,148.953
C03380=1183.330,23.233,-46.168,-179.706,5.847,148.953
C03381=1183.335,22.984,-46.153,-179.709,5.847,148.954
C03382=1183.340,22.734,-46.138,-179.711,5.846,148.955
C03383=1183.345,22.484,-46.124,-179.713,5.845,148.955
C03384=1183.350,22.235,-46.109,-179.716,5.845,148.956
C03385=1183.356,21.986,-46.095,-179.719,5.844,148.956
C03386=1183.360,21.736,-46.080,-179.721,5.843,148.957
C03387=1183.365,21.487,-46.065,-179.724,5.843,148.958
C03388=1183.370,21.237,-46.051,-179.727,5.842,148.958
C03389=1183.376,20.987,-46.036,-179.729,5.841,148.959
C03390=1183.380,20.738,-46.021,-179.732,5.840,148.959
C03391=1183.385,20.489,-46.007,-179.734,5.840,148.960
C03392=1183.390,20.239,-45.993,-179.736,5.839,148.961
C03393=1183.395,19.990,-45.978,-179.739,5.838,148.961
C03394=1183.401,19.740,-45.963,-179.742,5.838,148.962
C03395=1183.406,19.490,-45.949,-179.744,5.837,148.962
C03396=1183.410,19.241,-45.934,-179.746,5.837,148.963
C03397=1183.415,18.991,-45.919,-179.749,5.836,148.964
C03398=1183.421,18.742,-45.905,-179.752,5.836,148.964
C03399=1183.426,18.493,-45.891,-179.754,5.835,148.965
C03400=1183.431,18.243,-45.875,-179.757,5.834,148.966
C03401=1183.436,17.993,-45.861,-179.759,5.834,148.966
C03402=1183.441,17.744,-45.847,-179.762,5.832,148.967
C03403=1183.446,17.494,-45.833,-179.765,5.832,148.967
C03404=1183.451,17.244,-45.818,-179.767,5.831,148.968
C03405=1183.456,16.995,-45.803,-179.769,5.830,148.968
C03406=1183.461,16.746,-45.789,-179.772,5.830,148.969
C03407=1183.466,16.497,-45.775,-179.775,5.829,148.970
C03408=1183.471,16.247,-45.761,-179.777,5.828,148.970
C03409=1183.477,15.997,-45.746,-179.780,5.828,148.971
C03410=1183.481,15.748,-45.731,-179.782,5.828,148.972
C03411=1183.486,15.498,-45.717,-179.785,5.827,148.972
C03412=1183.491,15.248,-45.703,-179.787,5.826,148.973
C03413=1183.497,14.999,-45.689,-179.790,5.826,148.974
C03414=1183.502,14.750,-45.674,-179.792,5.825,148.974
C03415=1183.507,14.500,-45.660,-179.794,5.824,148.975
C03416=1183.512,14.250,-45.646,-179.797,5.824,148.975
C03417=1183.517,14.000,-45.631,-179.800,5.823,148.976
C03418=1183.522,13.751,-45.617,-179.802,5.823,148.976
C03419=1183.527,13.502,-45.603,-179.805,5.822,148.977
C03420=1183.532,13.253,-45.588,-179.807,5.822,148.978
C03421=1183.537,13.003,-45.574,-179.809,5.821,148.978
C03422=1183.542,12.753,-45.560,-179.812,5.820,148.979
C03423=1183.547,12.503,-45.545,-179.815,5.820,148.980
C03424=1183.552,12.254,-45.532,-179.817,5.819,148.980
C03425=1183.557,12.005,-45.517,-179.820,5.818,148.981
C03426=1183.562,11.755,-45.503,-179.822,5.818,148.981
C03427=1183.567,11.505,-45.489,-179.825,5.817,148.982
C03428=1183.572,11.256,-45.474,-179.828,5.816,148.983
C03429=1183.578,11.007,-45.461,-179.830,5.815,148.983
C03430=1183.583,10.757,-45.446,-179.833,5.815,148.984
C03431=1183.588,10.507,-45.432,-179.835,5.814,148.984
C03432=1183.593,10.257,-45.418,-179.838,5.813,148.985
C03433=1183.598,10.008,-45.404,-179.840,5.813,148.986
C03434=1183.603,9.759,-45.390,-179.843,5.812,148.987
C03435=1183.608,9.509,-45.375,-179.845,5.812,148.987
C03436=1183.613,9.259,-45.361,-179.848,5.811,148.988
C03437=1183.618,9.010,-45.347,-179.850,5.811,148.988
C03438=1183.624,8.760,-45.333,-179.853,5.810,148.989
C03439=1183.628,8.511,-45.320,-179.855,5.809,148.989
C03440=1183.633,8.261,-45.306,-179.858,5.809,148.990
C03441=1183.638,8.012,-45.292,-179.860,5.808,148.991
C03442=1183.643,7.762,-45.277,-179.863,5.808,148.991
C03443=1183.648,7.512,-45.263,-179.865,5.807,148.992
C03444=1183.653,7.263,-45.249,-179.868,5.807,148.993
C03445=1183.659,7.014,-45.235,-179.870,5.806,148.993
C03446=1183.664,6.764,-45.221,-179.873,5.805,148.994
C03447=1183.668,6.514,-45.208,-179.876,5.805,148.995
C03448=1183.674,6.265,-45.194,-179.878,5.804,148.995
C03449=1183.679,6.015,-45.179,-179.880,5.803,148.996
C03450=1183.684,5.766,-45.165,-179.883,5.803,148.996
C03451=1183.689,5.517,-45.151,-179.886,5.802,148.997
C03452=1183.694,5.267,-45.137,-179.888,5.802,148.997
C03453=1183.700,5.017,-45.123,-179.890,5.801,148.998
C03454=1183.704,4.768,-45.110,-179.893,5.801,148.999
C03455=1183.709,4.518,-45.096,-179.895,5.800,148.999
C03456=1183.714,4.268,-45.082,-179.898,5.799,149.000
C03457=1183.720,4.018,-45.068,-179.901,5.799,149.001
C03458=1183.725,3.769,-45.054,-179.903,5.798,149.001
C03459=1183.729,3.520,-45.040,-179.905,5.798,149.002
C03460=1183.735,3.271,-45.026,-179.908,5.797,149.003
C03461=1183.740,3.020,-45.013,-179.911,5.797,149.003
C03462=1183.746,2.751,-44.998,-179.913,5.796,149.004
C03463=1183.751,2.482,-44.982,-179.916,5.795,149.004
C03464=1183.757,2.213,-44.968,-179.918,5.795,149.005
C03465=1183.762,1.944,-44.953,-179.921,5.794,149.006
C03466=1183.767,1.694,-44.940,-179.924,5.794,149.006
C03467=1183.772,1.444,-44.925,-179.926,5.793,149.007
C03468=1183.777,1.195,-44.911,-179.928,5.793,149.008
C03469=1183.783,0.945,-44.898,-179.931,5.792,149.008
C03470=1183.787,0.696,-44.885,-179.934,5.792,149.009
C03471=1183.792,0.447,-44.870,-179.936,5.791,149.010
C03472=1183.798,0.196,-44.857,-179.938,5.790,149.010
C03473=1183.802,-0.052,-44.843,-179.941,5.790,149.011
C03474=1183.808,-0.303,-44.830,-179.944,5.789,149.011
C03475=1183.813,-0.552,-44.816,-179.946,5.788,149.012
C03476=1183.818,-0.802,-44.802,-179.949,5.788,149.013
C03477=1183.823,-1.052,-44.789,-179.951,5.788,149.013
C03478=1183.828,-1.301,-44.775,-179.954,5.787,149.014
C03479=1183.833,-1.551,-44.761,-179.956,5.786,149.014
C03480=1183.838,-1.800,-44.748,-179.959,5.786,149.015
C03481=1183.843,-2.049,-44.734,-179.961,5.785,149.016
C03482=1183.849,-2.299,-44.720,-179.963,5.785,149.016
C03483=1183.853,-2.548,-44.707,-179.966,5.785,149.017
C03484=1183.859,-2.799,-44.693,-179.968,5.784,149.018
C03485=1183.864,-3.048,-44.679,-179.971,5.784,149.018
C03486=1183.869,-3.298,-44.666,-179.973,5.783,149.019
C03487=1183.874,-3.547,-44.652,-179.976,5.782,149.020
C03488=1183.879,-3.797,-44.639,-179.978,5.782,149.020
C03489=1183.884,-4.046,-44.626,-179.981,5.781,149.021
C03490=1183.890,-4.296,-44.612,-179.983,5.781,149.021
C03491=1183.894,-4.545,-44.599,-179.986,5.780,149.022
C03492=1183.900,-4.795,-44.585,-179.989,5.780,149.023
C03493=1183.904,-5.044,-44.572,-179.991,5.779,149.023
C03494=1183.910,-5.294,-44.558,-179.993,5.778,149.024
C03495=1183.915,-5.544,-44.544,-179.996,5.778,149.025
C03496=1183.920,-5.793,-44.531,-179.999,5.777,149.025
C03497=1183.925,-6.043,-44.517,179.999,5.777,149.026
C03498=1183.930,-6.292,-44.504,179.996,5.776,149.026
C03499=1183.935,-6.543,-44.491,179.994,5.776,149.027
C03500=1183.940,-6.791,-44.478,179.992,5.776,149.028
C03501=1183.945,-7.042,-44.464,179.990,5.775,149.028
C03502=1183.951,-7.291,-44.450,179.987,5.775,149.029
C03503=1183.955,-7.541,-44.437,179.984,5.774,149.030
C03504=1183.961,-7.790,-44.424,179.982,5.773,149.030
C03505=1183.965,-8.040,-44.410,179.979,5.773,149.031
C03506=1183.971,-8.289,-44.397,179.977,5.772,149.032
C03507=1183.976,-8.539,-44.384,179.975,5.772,149.032
C03508=1183.981,-8.788,-44.370,179.972,5.771,149.033
C03509=1183.986,-9.038,-44.358,179.969,5.771,149.033
C03510=1183.992,-9.288,-44.344,179.967,5.770,149.034
C03511=1183.997,-9.537,-44.331,179.964,5.769,149.035
C03512=1184.002,-9.787,-44.317,179.962,5.769,149.035
C03513=1184.007,-10.036,-44.305,179.960,5.769,149.036
C03514=1184.012,-10.286,-44.290,179.958,5.768,149.036
C03515=1184.017,-10.535,-44.278,179.955,5.768,149.037
C03516=1184.022,-10.785,-44.265,179.952,5.768,149.038
C03517=1184.027,-11.034,-44.251,179.950,5.767,149.038
C03518=1184.032,-11.284,-44.238,179.947,5.766,149.039
C03519=1184.037,-11.534,-44.225,179.945,5.766,149.040
C03520=1184.043,-11.783,-44.212,179.942,5.765,149.040
C03521=1184.048,-12.033,-44.198,179.939,5.765,149.041
C03522=1184.053,-12.282,-44.185,179.937,5.764,149.041
C03523=1184.058,-12.533,-44.172,179.935,5.764,149.042
C03524=1184.063,-12.782,-44.159,179.933,5.764,149.043
C03525=1184.068,-13.031,-44.146,179.930,5.763,149.043
C03526=1184.073,-13.281,-44.132,179.928,5.763,149.044
C03527=1184.078,-13.530,-44.120,179.925,5.762,149.045
C03528=1184.083,-13.781,-44.106,179.922,5.762,149.045
C03529=1184.089,-14.030,-44.093,179.920,5.761,149.046
C03530=1184.094,-14.279,-44.081,179.918,5.760,149.047
C03531=1184.099,-14.529,-44.066,179.915,5.760,149.047
C03532=1184.104,-14.778,-44.054,179.913,5.759,149.048
C03533=1184.108,-15.028,-44.041,179.911,5.759,149.048
C03534=1184.114,-15.278,-44.028,179.908,5.759,149.049
C03535=1184.119,-15.527,-44.015,179.905,5.758,149.050
C03536=1184.125,-15.778,-44.002,179.903,5.758,149.050
C03537=1184.130,-16.027,-43.989,179.901,5.757,149.051
C03538=1184.135,-16.276,-43.976,179.898,5.757,149.052
C03539=1184.140,-16.526,-43.962,179.895,5.756,149.052
C03540=1184.145,-16.775,-43.949,179.893,5.755,149.053
C03541=1184.150,-17.025,-43.937,179.890,5.755,149.053
C03542=1184.155,-17.275,-43.923,179.888,5.755,149.054
C03543=1184.160,-17.524,-43.911,179.886,5.754,149.055
C03544=1184.165,-17.774,-43.898,179.883,5.754,149.055
C03545=1184.170,-18.024,-43.885,179.881,5.754,149.056
C03546=1184.176,-18.273,-43.872,179.878,5.753,149.057
C03547=1184.181,-18.522,-43.859,179.876,5.752,149.057
C03548=1184.186,-18.773,-43.846,179.873,5.752,149.058
C03549=1184.191,-19.022,-43.833,179.871,5.751,149.059
C03550=1184.197,-19.271,-43.821,179.869,5.752,149.059
C03551=1184.201,-19.521,-43.808,179.866,5.751,149.060
C03552=1184.206,-19.771,-43.795,179.864,5.750,149.060
C03553=1184.212,-20.020,-43.782,179.861,5.750,149.061
C03554=1184.217,-20.270,-43.769,179.859,5.749,149.062
C03555=1184.222,-20.520,-43.756,179.856,5.749,149.062
C03556=1184.227,-20.769,-43.744,179.854,5.748,149.063
C03557=1184.233,-21.019,-43.730,179.852,5.749,149.064
C03558=1184.237,-21.269,-43.717,179.849,5.748,149.064
C03559=1184.242,-21.518,-43.705,179.847,5.747,149.065
C03560=1184.247,-21.767,-43.692,179.844,5.747,149.066
C03561=1184.253,-22.018,-43.679,179.841,5.746,149.066
C03562=1184.258,-22.267,-43.666,179.839,5.745,149.067
C03563=1184.263,-22.516,-43.654,179.837,5.745,149.067
C03564=1184.268,-22.766,-43.642,179.834,5.745,149.068
C03565=1184.273,-23.016,-43.629,179.832,5.745,149.069
C03566=1184.279,-23.286,-43.615,179.830,5.744,149.069
C03567=1184.284,-23.555,-43.601,179.827,5.744,149.070
C03568=1184.290,-23.825,-43.587,179.824,5.743,149.071
C03569=1184.296,-24.094,-43.573,179.822,5.743,149.071
C03570=1184.300,-24.344,-43.561,179.819,5.742,149.072
C03571=1184.305,-24.594,-43.548,179.816,5.742,149.073
C03572=1184.311,-24.844,-43.535,179.814,5.741,149.073
C03573=1184.317,-25.093,-43.523,179.811,5.741,149.074
C03574=1184.322,-25.343,-43.510,179.809,5.740,149.075
C03575=1184.326,-25.593,-43.497,179.807,5.740,149.075
C03576=1184.331,-25.842,-43.485,179.805,5.740,149.076
C03577=1184.336,-26.091,-43.472,179.802,5.739,149.076
C03578=1184.342,-26.341,-43.460,179.799,5.739,149.077
C03579=1184.346,-26.591,-43.447,179.797,5.738,149.078
C03580=1184.352,-26.841,-43.435,179.794,5.737,149.078
C03581=1184.357,-27.090,-43.421,179.792,5.738,149.079
C03582=1184.363,-27.340,-43.410,179.790,5.737,149.080
C03583=1184.368,-27.589,-43.397,179.788,5.736,149.080
C03584=1184.372,-27.839,-43.384,179.785,5.736,149.081
C03585=1184.378,-28.089,-43.371,179.782,5.736,149.082
C03586=1184.383,-28.339,-43.359,179.780,5.735,149.082
C03587=1184.388,-28.588,-43.347,179.778,5.735,149.083
C03588=1184.393,-28.837,-43.334,179.775,5.735,149.083
C03589=1184.398,-29.087,-43.322,179.773,5.734,149.084
C03590=1184.403,-29.337,-43.309,179.770,5.733,149.085
C03591=1184.408,-29.587,-43.297,179.768,5.733,149.085
C03592=1184.413,-29.836,-43.284,179.765,5.732,149.086
C03593=1184.419,-30.086,-43.272,179.763,5.733,149.087
C03594=1184.424,-30.335,-43.260,179.761,5.732,149.087
C03595=1184.429,-30.584,-43.247,179.758,5.732,149.088
C03596=1184.434,-30.835,-43.235,179.756,5.731,149.089
C03597=1184.439,-31.084,-43.222,179.753,5.730,149.089
C03598=1184.444,-31.334,-43.210,179.751,5.731,149.090
C03599=1184.450,-31.584,-43.198,179.749,5.730,149.090
C03600=1184.455,-31.833,-43.185,179.746,5.730,149.091
C03601=1184.460,-32.083,-43.173,179.744,5.729,149.092
C03602=1184.465,-32.332,-43.161,179.741,5.728,149.092
C03603=1184.470,-32.582,-43.148,179.739,5.729,149.093
C03604=1184.475,-32.832,-43.136,179.736,5.728,149.094
C03605=1184.480,-33.082,-43.123,179.734,5.728,149.094
C03606=1184.486,-33.331,-43.111,179.732,5.727,149.095
C03607=1184.491,-33.581,-43.099,179.729,5.727,149.096
C03608=1184.496,-33.831,-43.087,179.727,5.727,149.096
C03609=1184.502,-34.080,-43.074,179.725,5.726,149.097
C03610=1184.507,-34.329,-43.062,179.722,5.726,149.097
C03611=1184.512,-34.579,-43.050,179.719,5.725,149.098
C03612=1184.517,-34.829,-43.037,179.717,5.724,149.099
C03613=1184.523,-35.079,-43.025,179.715,5.725,149.099
C03614=1184.528,-35.328,-43.013,179.712,5.724,149.100
C03615=1184.533,-35.579,-43.000,179.710,5.724,149.100
C03616=1184.538,-35.828,-42.988,179.708,5.723,149.101
C03617=1184.542,-36.077,-42.977,179.705,5.723,149.102
C03618=1184.548,-36.327,-42.964,179.703,5.723,149.103
C03619=1184.553,-36.577,-42.952,179.701,5.722,149.103
C03620=1184.558,-36.826,-42.939,179.698,5.722,149.104
C03621=1184.563,-37.076,-42.928,179.695,5.721,149.104
C03622=1184.569,-37.325,-42.915,179.693,5.721,149.105
C03623=1184.574,-37.575,-42.903,179.691,5.721,149.106
C03624=1184.579,-37.825,-42.891,179.688,5.720,149.106
C03625=1184.585,-38.074,-42.879,179.686,5.720,149.107
C03626=1184.589,-38.324,-42.867,179.684,5.719,149.108
C03627=1184.594,-38.573,-42.855,179.681,5.719,149.108
C03628=1184.600,-38.823,-42.843,179.679,5.719,149.109
C03629=1184.605,-39.073,-42.831,179.676,5.719,149.110
C03630=1184.610,-39.323,-42.818,179.674,5.718,149.110
C03631=1184.616,-39.573,-42.806,179.671,5.717,149.111
C03632=1184.620,-39.822,-42.794,179.669,5.718,149.111
C03633=1184.626,-40.071,-42.783,179.667,5.717,149.112
C03634=1184.631,-40.321,-42.771,179.664,5.716,149.113
C03635=1184.636,-40.571,-42.758,179.662,5.716,149.113
C03636=1184.642,-40.821,-42.746,179.659,5.716,149.114
C03637=1184.646,-41.070,-42.735,179.657,5.716,149.115
C03638=1184.651,-41.320,-42.722,179.655,5.715,149.115
C03639=1184.657,-41.570,-42.710,179.652,5.715,149.116
C03640=1184.662,-41.820,-42.699,179.650,5.714,149.116
C03641=1184.667,-42.069,-42.686,179.648,5.714,149.117
C03642=1184.672,-42.318,-42.675,179.645,5.714,149.118
C03643=1184.678,-42.568,-42.663,179.643,5.713,149.119
C03644=1184.683,-42.818,-42.650,179.640,5.712,149.119
C03645=1184.688,-43.068,-42.638,179.638,5.713,149.120
C03646=1184.693,-43.317,-42.627,179.636,5.712,149.120
C03647=1184.698,-43.567,-42.615,179.633,5.712,149.121
C03648=1184.703,-43.817,-42.603,179.631,5.711,149.122
